// SIMATIC STEP 7 (V5.x) project GYPSUM
// CPU: CPU 317-2 DP
// station: P_ADR_BUS
// station: _S7H_BUSSYSTEM_CT
// station: Hardware
// station: SIMATIC 300(1)
// program: S7 Program(1)

SYMBOL_TABLE
"GROUPS"	DB 15	DB 15
"ROUTES"	DB 16	DB 16
"HMI"	DB 20	DB 20	// HMI
"RECEPT"	DB 21	DB 21
"G00_MILL_GYPSUM"	DB 30	FB 103	// Mill Gypsum
"G01_BIN_LOAD"	DB 31	FB 103	// 311BI100 Loading
"G02_EFILER"	DB 32	FB 103	// ElectroFilter Group
"G03_FRESH_GYPSUM"	DB 33	FB 103	// Fresh Gypsum
"G04_BOILER1"	DB 34	FB 103	// Boiler 1 Group
"G05_WEIGHT_PALLET"	DB 35	FB 103	// Weight Pallet
"G06_DISCHARGE"	DB 36	FB 103	// Discharge Group
"G07_BOILER2"	DB 37	FB 103	// G07 Boiler 2
"G08_BOILER3"	DB 38	FB 103	// G08 Boiler 3
"G17_DUMMY_LOCAL"	DB 47	FB 103
"G18_DUMMY_MANUAL"	DB 48	FB 103
"G19_DUMMY_ASTR"	DB 49	FB 103
"REG_T_BeforeSeparator"	DB 51	FB 41	// Temperature Regler Before Separator
"REG_DiffP_AfterSeparator"	DB 52	FB 41	// Diff Pressure Regler After Separator
"REG_Curr_CrusherMD140"	DB 53	FB 41	// Current Regler Crusher MD140
"REG_DiffP_Boiler3"	DB 54	FB 41	// Diff Pressure Regler Boiler  3
"REG_DiffP_Boiler1"	DB 55	FB 41	// Diff Pressure Regler Boiler 1
"REG_DiffP_Boiler2"	DB 56	FB 41	// Diff Pressure Regler Boiler 2
"Weight351BI100"	DB 61	FB 310	// Weight351BI100
"Weight351BI200"	DB 62	FB 310	// Weight351BI200
"Weight351BI300"	DB 63	FB 310	// Weight 351BI300 Fresh Gypsum
"Weight352BI100"	DB 64	FB 310	// Weight352BI100
"Weight352BI200"	DB 65	FB 310
"Weight352BI300"	DB 66	FB 310	// Weight352BI300
"Weight351BI130"	DB 67	FB 310	// Weight351BI130
"Weight351BI230"	DB 68	FB 310	// Weight351BI230
"Weight351BI330"	DB 69	FB 310	// Weight351BI330
"Boiler 1"	DB 70	FB 310	// Boler 1
"Boiler 2"	DB 71	FB 310	// Boiler 2
"Boiler 3"	DB 72	FB 310	// Boiler 3
"411DC100N01T01"	DB 101	FB 101	// Temperature Before Crusher
"411DC100N02P01"	DB 102	FB 101	// Pressure Before Crusher
"411DC100N03T02"	DB 103	FB 101	// Temperature After Crusher
"411DC100N04P02"	DB 104	FB 101	// Pressure After Crusher
"351BR300N06T04"	DB 105	FB 101	// Temperature Hot Air
"351BR300N07P03"	DB 106	FB 101	// Pressure Hot Air
"351BI100N01T01"	DB 107	FB 101	// Temperature In 351BI100
"351BI200N01T01"	DB 108	FB 101	// Temperature In 351BI200
"351BI300N01T01"	DB 109	FB 101	// Temperature In 351BI300
"351BR100N01T01"	DB 110	FB 101	// Temperature In Boiler 1 Top
"351BR100N02T02"	DB 111	FB 101	// Temperature In Boiler 1 Bottom
"351BR100N03P01"	DB 112	FB 101	// Pressure In Boiler 1 Bottom
"351BR200N01T01"	DB 113	FB 101	// Temperature In Boiler 2 Top
"351BR200N02T02"	DB 114	FB 101	// Temperature In Boiler 2 Bottom
"351BR200N03P01"	DB 115	FB 101	// Pressure In Boiler 2 Bottom
"351BR300N01T01"	DB 116	FB 101	// Temperature In Biler 3 Top
"351BR300N02T02"	DB 117	FB 101	// Temperature In Boiler 3 Bottom
"351BR300N03P01"	DB 118	FB 101	// Pressure In Boiler 3 Bottom
"331EP100N01P01"	DB 119	FB 101	// Pressure Before EFilter
"351BI100N02W01"	DB 120	FB 101	// Bin Weight 351BI100
"351BI200N02W01"	DB 121	FB 101	// Bin Weight 351BI200
"351BI300N02W01"	DB 122	FB 101	// Bin Weight 351BI300
"352BI100N01W01"	DB 123	FB 101	// Bin Weight 352BI100
"352BI200N01W01"	DB 124	FB 101	// Bin Weight 352BI200
"352BI300N01W01"	DB 125	FB 101	// Bin Weight 352BI300
"351BI130N01W01"	DB 126	FB 101	// Bin Weight 351BI130
"351BI230N01W01"	DB 127	FB 101	// Bin Weight 351BI230
"351BI330N01W01"	DB 128	FB 101	// Bin Weight 351BI330
"331EP100N02T01"	DB 129	FB 101	// Temperature Before EFilter
"331EP100N03T02"	DB 130	FB 101	// Temperature After EFilter
"331EP100N04P02"	DB 131	FB 101	// Pressure After EFilter
"331LD391Z01"	DB 132	FB 101	// Position Gate
"331LD392Z01"	DB 133	FB 101	// Position Gate
"411CN101N01P01"	DB 134	FB 101	// Pressure Before Cyclone
"411CN101N02T01"	DB 135	FB 101	// Temperature Before Cyclone
"411CN101N03P02"	DB 136	FB 101	// Pressure After Cyclone
"411CN101N04T02"	DB 137	FB 101	// Temperature After Cyclone
"411CN103N01P01"	DB 138	FB 101	// Pressure After Cyclone
"411CN103N02T01"	DB 139	FB 101	// Temperature After Cyclone
"351BR100N04T03"	DB 140	FB 101	// Temperature in Burner Boiler 1
"351BR100N05P02"	DB 141	FB 101	// Pressure In Burner Boiler 1
"351BR200N04T03"	DB 142	FB 101	// Temperature In Boiler 2
"351BR200N05P02"	DB 143	FB 101	// Pressure In Burner Boiler 2
"351BR300N04T03"	DB 144	FB 101	// Temperature In Burner Boiler 3
"351BR300N05P02"	DB 145	FB 101	// Pressure In Burner Boiler 3
"411SR150N03T02"	DB 146	FB 101	// Temperature Before Separator (Bearing)
"SPARE_AI47"	DB 147	FB 101
"143CV100SI01"	DB 148	FB 101	// Speed Chain Conveyor CV100
"143CV100UA01"	DB 149	FB 101	// Current Chain Conveyor CV100
"143BC200SI01"	DB 150	FB 101	// Speed Belt Conveyor BC200
"143BC200UA01"	DB 151	FB 101	// Current Belt Conveyor BC200
"331FN401SI01"	DB 152	FB 101	// Speed EFilter Fan FN401
"331FN401UA01"	DB 153	FB 101	// Current EFilter Fan FN401
"311TF150SI01"	DB 154	FB 101	// Speed Table Feeder TF150
"311TF150UA01"	DB 155	FB 101	// Current Table Feeder TF150
"411MD140SI01"	DB 156	FB 101	// Speed Crusher MD140
"411MD140UA01"	DB 157	FB 101	// Current Crusher MD140
"411MD152SI01"	DB 158	FB 101	// Speed Separator MD152
"411MD152UA01"	DB 159	FB 101	// Current Separator MD152
"351SC120SI01"	DB 160	FB 101	// Speed Screw Conveyor SC120
"351SC120UA01"	DB 161	FB 101	// Current Screw Conveyor SC120
"351SC220SI01"	DB 162	FB 101	// Speed Screw Conveyor SC220
"351SC220UA01"	DB 163	FB 101	// Current Screw Conveyor SC220
"351SC320SI01"	DB 164	FB 101	// Speed Screw Conveyor SC320
"351SC320UA01"	DB 165	FB 101	// Current Screw Conveyor SC320
"361SC140SI01"	DB 166	FB 101	// Speed Screw Conveyor SC140
"361SC140UA01"	DB 167	FB 101	// Current Screw Conveyor SC140
"351BR100N06T04"	DB 168	FB 101	// Temperature Hot Air From Boiler 1
"351BR200N06T04"	DB 169	FB 101	// Temperature Hot Air From Boiler 2
"351BR300N08T04"	DB 170	FB 101	// Temperature Hot Air From Boiler 3
"351SD101N01Z01"	DB 171	FB 101
"351SD102N01Z01"	DB 172	FB 101
"351SD103N01Z01"	DB 173	FB 101
"351SD104N01Z01"	DB 174	FB 101
"351Sd105N01Z01"	DB 175	FB 101
"100CP100N01P01"	DB 176	FB 101	// Pressure After Compressor
"BE120_CUR"	DB 177	FB 101	// BE120 Current AL
"SPARE_AI78"	DB 178	FB 101
"SPARE_AI79"	DB 179	FB 101
"SPARE_AI80"	DB 180	FB 101
"SPARE_AI81"	DB 181	FB 101
"SPARE_AI82"	DB 182	FB 101
"SPARE_AI83"	DB 183	FB 101
"SPARE_AI84"	DB 184	FB 101
"SPARE_AI85"	DB 185	FB 101
"SPARE_AI86"	DB 186	FB 101
"SPARE_AI87"	DB 187	FB 101
"SPARE_AI88"	DB 188	FB 101
"SPARE_AI89"	DB 189	FB 101
"SPARE_AI90"	DB 190	FB 101
"SPARE_AI91"	DB 191	FB 101
"SPARE_AI92"	DB 192	FB 101
"SPARE_AI93"	DB 193	FB 101
"SPARE_AI94"	DB 194	FB 101
"SPARE_AI95"	DB 195	FB 101
"SPARE_AI96"	DB 196	FB 101
"SPARE_AI97"	DB 197	FB 101
"SPARE_AI98"	DB 198	FB 101
"SPARE_AI99"	DB 199	FB 101
"SPARE_UNIMOTOR01"	DB 201	FB 110
"143BF120"	DB 202	FB 110	// Filter Control
"351VI110"	DB 203	FB 110	// Vibrator
"351VI210"	DB 204	FB 110	// Vibrator
"351VI310"	DB 205	FB 110	// Vibrator
"352VI110"	DB 206	FB 110	// Vibrator
"352VI111"	DB 207	FB 110	// Vibrator
"352VI210"	DB 208	FB 110	// Vibrator
"352VI211"	DB 209	FB 110	// Vibrator
"352VI310"	DB 210	FB 110	// Vibrator
"352VI311"	DB 211	FB 110	// Vibrator
"EP100P1"	DB 212	FB 110	// EFilter Pole 1
"EP100P2"	DB 213	FB 110	// EFilter Pole   2
"SPARE_UNIMOTOR14"	DB 214	FB 110
"SPARE_UNIMOTOR15"	DB 215	FB 110
"SPARE_UNIMOTOR16"	DB 216	FB 110
"SPARE_UNIMOTOR17"	DB 217	FB 110
"SPARE_UNIMOTOR18"	DB 218	FB 110
"SPARE_UNIMOTOR19"	DB 219	FB 110
"SPARE_UNIMOTOR20"	DB 220	FB 110
"411SD311"	DB 251	FB 102	// Gate Gypsum To Pneumatic Pump
"412SD321"	DB 252	FB 102	// Gate Gypsum To Screw Conveyor
"411SD331"	DB 253	FB 102	// Gate Weight 351BI100 Inlet
"411SD332"	DB 254	FB 102	// Gate Weight 351BI200 Inlet
"411SD333"	DB 255	FB 102	// Gate Weight 351BI300 Inlet
"351SD140"	DB 256	FB 102	// Gate Boiler 1 Outlet
"351SD141"	DB 257	FB 102	// Gate Boiler 1 Outlet
"352SD120"	DB 258	FB 102	// Gate Weight 352BI100 Outlet
"352SD121"	DB 259	FB 102	// Gate Weight 352BI100 Outlet
"351SD240"	DB 260	FB 102	// Gate Boiler 2 Outlet
"351SD241"	DB 261	FB 102	// Gate Boiler 2 Outlet
"352SD220"	DB 262	FB 102	// Gate Weight 352BI200 Outlet
"352SD221"	DB 263	FB 102	// Gate Weight 352BI200 Outlet
"351SD340"	DB 264	FB 102	// Gate Boiler 3 Outlet
"351SD341"	DB 265	FB 102	// Gate Boiler 3 Outlet
"352SD320"	DB 266	FB 102	// Gate Weight 352BI300 Outlet
"352SD321"	DB 267	FB 102	// Gate Weight 352BI300 Outlet
"361SD170"	DB 268	FB 102	// Gate 371BI500 Inlet
"361SD171"	DB 269	FB 102	// Gate 371BI100 Inlet
"361SD172"	DB 270	FB 102	// Gate 371BI100 Inlet
"361SD173"	DB 271	FB 102	// Gate 371BI200 Inlet
"361SD174"	DB 272	FB 102	// Gate 371B200 Inlet
"361SD175"	DB 273	FB 102	// Gate 371BI300 Inlet
"361SD176"	DB 274	FB 102	// Gate 371BI300 Inlet
"361SD177"	DB 275	FB 102	// Gate 371BI400 Inlet
"351BV031"	DB 276	FB 102	// Valve Aqua To Boiler 1
"351BV032"	DB 277	FB 102	// Valve Aqua To Boiler 2
"351BV033"	DB 278	FB 102	// Valve Aqua To Boiler 3
"351SD135"	DB 279	FB 102	// Gate Weight 351BI130 Inlet
"351SD235"	DB 280	FB 102	// Gate Weight 351BI230 Inlet
"351SD335"	DB 281	FB 102	// Gate Weight 351BI330 Inlet
"411BV151"	DB 282	FB 102	// Valve Separator Aspiration
"SPARE_VALVE33"	DB 283	FB 102
"351SD106"	DB 284	FB 102	// Gate Boiler 1 Outlet Hot Air
"351SD107"	DB 285	FB 102	// Gate Boiler 1 Outlet
"351SD108"	DB 286	FB 102	// Gate Boiler 3 Outlet
"351SD109"	DB 287	FB 102	// Gate Hot Air To Gypsum Line
"SPARE_VALVE38"	DB 288	FB 102
"SPARE_VALVE39"	DB 289	FB 102
"SPARE_VALVE40"	DB 290	FB 102
"SPARE_UMOTSC01"	DB 301	FB 134
"143VF150"	DB 302	FB 134	// Vibrating Din
"143BC160"	DB 303	FB 134	// Belt Conveyor
"SPARE_UMOTSC04"	DB 304	FB 134
"143RB250"	DB 305	FB 134	// Crusher
"143BE300"	DB 306	FB 134	// Elevator
"143FN122"	DB 307	FB 134	// Filter Fan
"311RF200"	DB 308	FB 134	// Rotary Feeder
"41FN101"	DB 309	FB 134	// Fan Crusher Drive Cooling
"411RF201"	DB 310	FB 134	// Rotary Feeder
"411RF304"	DB 311	FB 134	// Rotary Feeder
"411SC322"	DB 312	FB 134	// Screw Conveyor
"331VI201"	DB 313	FB 134	// Filter Rapping 1
"331VI202"	DB 314	FB 134	// Filter Rapping 2
"331VI203"	DB 315	FB 134	// Filter Rapping 3
"331VI204"	DB 316	FB 134	// Filter Rapping 4
"331RF301"	DB 317	FB 134	// Rotary Feeder
"331RF302"	DB 318	FB 134	// Rotary Feeder
"331RF303"	DB 319	FB 134	// Rotary Feeder
"331SC351"	DB 320	FB 134	// Screw Conveyor
"411RF314"	DB 321	FB 134	// Rotary Feeder
"361SC150"	DB 322	FB 134	// Screw Conveyor
"SPARE_UMOTSC23"	DB 323	FB 134
"411PP312"	DB 324	FB 134	// Pneumatic Pump
"SPARE_UMOTSC25"	DB 325	FB 134
"SPARE_UMOTSC26"	DB 326	FB 134
"351AG130"	DB 327	FB 134	// Mixer 1
"351AG230"	DB 328	FB 134	// Mixer 2
"351AG330"	DB 329	FB 134	// Mixer 3
"361SC110"	DB 330	FB 134	// Screw Conveyor
"361SC111"	DB 331	FB 134	// Screw Conveyor
"361BE120"	DB 332	FB 134	// Elevator
"361SC130"	DB 333	FB 134	// Screw Conveyor
"SPARE_UMOTSC34"	DB 334	FB 134
"361SC141"	DB 335	FB 134	// Screw Conveyor
"SPARE_UMOTSC36"	DB 336	FB 134
"361SC160"	DB 337	FB 134	// Screw Conveyor
"341RF101"	DB 338	FB 134	// Rotary Feeder
"SPARE_UMOTSC39"	DB 339	FB 134	// Spare
"411FN200"	DB 340	FB 134	// Fan Hot Air To Crusher
"351AG050"	DB 341	FB 134	// Mixer
"351SP100"	DB 342	FB 134	// Pump
"SPARE_UMOTSC43"	DB 343	FB 134
"SPARE_UMOTSC44"	DB 344	FB 134
"SPARE_UMOTSC45"	DB 345	FB 134
"SPARE_UMOTSC46"	DB 346	FB 134
"SPARE_UMOTSC47"	DB 347	FB 134
"SPARE_UMOTSC48"	DB 348	FB 134
"SPARE_UMOTSC49"	DB 349	FB 134
"SPARE_UMOTSC50"	DB 350	FB 134
"SPARE_UMOTSC51"	DB 351	FB 134
"SPARE_UMOTSC52"	DB 352	FB 134
"SPARE_UMOTSC53"	DB 353	FB 134
"SPARE_UMOTSC54"	DB 354	FB 134
"SPARE_UMOTSC55"	DB 355	FB 134
"SPARE_UMOTSC56"	DB 356	FB 134
"SPARE_UMOTSC57"	DB 357	FB 134
"SPARE_UMOTSC58"	DB 358	FB 134
"SPARE_UMOTSC59"	DB 359	FB 134
"SPARE_UMOTSC60"	DB 360	FB 134
"SPARE_UMOTSC61"	DB 361	FB 134
"SPARE_UMOTSC62"	DB 362	FB 134
"SPARE_UMOTSC63"	DB 363	FB 134
"SPARE_UMOTSC64"	DB 364	FB 134
"SPARE_UMOTSC65"	DB 365	FB 134
"SPARE_UMOTSC66"	DB 366	FB 134
"SPARE_UMOTSC67"	DB 367	FB 134
"SPARE_UMOTSC68"	DB 368	FB 134
"SPARE_UMOTSC69"	DB 369	FB 134
"SPARE_UMOTSC70"	DB 370	FB 134
"SPARE_UMOTSC71"	DB 371	FB 134
"SPARE_UMOTSC72"	DB 372	FB 134
"SPARE_UMOTSC73"	DB 373	FB 134
"SPARE_UMOTSC74"	DB 374	FB 134
"SPARE_UMOTSC75"	DB 375	FB 134
"SPARE_UMOTSC76"	DB 376	FB 134
"SPARE_UMOTSC77"	DB 377	FB 134
"SPARE_UMOTSC78"	DB 378	FB 134
"SPARE_UMOTSC79"	DB 379	FB 134
"SPARE_UMOTSC80"	DB 380	FB 134
"SPARE_UMOTSC81"	DB 381	FB 134
"SPARE_UMOTSC82"	DB 382	FB 134
"SPARE_UMOTSC83"	DB 383	FB 134
"SPARE_UMOTSC84"	DB 384	FB 134
"SPARE_UMOTSC85"	DB 385	FB 134
"SPARE_UMOTSC86"	DB 386	FB 134
"SPARE_UMOTSC87"	DB 387	FB 134
"SPARE_UMOTSC88"	DB 388	FB 134
"SPARE_UMOTSC89"	DB 389	FB 134
"SPARE_UMOTSC90"	DB 390	FB 134
"SPARE_UMOTSC91"	DB 391	FB 134
"SPARE_UMOTSC92"	DB 392	FB 134
"SPARE_UMOTSC93"	DB 393	FB 134
"SPARE_UMOTSC94"	DB 394	FB 134
"SPARE_UMOTSC95"	DB 395	FB 134
"SPARE_UMOTSC96"	DB 396	FB 134
"SPARE_UMOTSC97"	DB 397	FB 134
"SPARE_UMOTSC98"	DB 398	FB 134
"SPARE_UMOTSC99"	DB 399	FB 134
"331LD391_SPARE"	DB 401	FB 136	// Gate Filter Fan
"331LD392_SPARE"	DB 402	FB 136	// Gate Filter Fan
"SPARE_AGATESC03"	DB 403	FB 136
"SPARE_AGATESC04"	DB 404	FB 136
"SPARE_AGATESC05"	DB 405	FB 136
"SPARE_AGATESC06"	DB 406	FB 136
"SPARE_AGATESC07"	DB 407	FB 136
"SPARE_AGATESC08"	DB 408	FB 136
"SPARE_AGATESC09"	DB 409	FB 136
"SPARE_AGATESC10"	DB 410	FB 136
"SPARE_GATESC01"	DB 451	FB 135
"SPARE_GATESC02"	DB 452	FB 135
"SPARE_GATESC03"	DB 453	FB 135
"SPARE_GATESC04"	DB 454	FB 135
"SPARE_GATESC05"	DB 455	FB 135
"SPARE_GATESC06"	DB 456	FB 135
"SPARE_GATESC07"	DB 457	FB 135
"SPARE_GATESC08"	DB 458	FB 135
"SPARE_GATESC09"	DB 459	FB 135
"SPARE_GATESC10"	DB 460	FB 135
"SPARE_BIMOTSC01"	DB 501	FB 139
"SPARE_BIMOTSC02"	DB 502	FB 139
"SPARE_BIMOTSC03"	DB 503	FB 139
"SPARE_BIMOTSC04"	DB 504	FB 139
"SPARE_BIMOTSC05"	DB 505	FB 139
"SPARE_BIMOTSC06"	DB 506	FB 139
"SPARE_BIMOTSC07"	DB 507	FB 139
"SPARE_BIMOTSC08"	DB 508	FB 139
"SPARE_BIMOTSC09"	DB 509	FB 139
"SPARE_BIMOTSC10"	DB 510	FB 139
"SPARE_BIMOTOR01"	DB 551	FB 109
"SPARE_BIMOTOR02"	DB 552	FB 109
"SPARE_BIMOTOR03"	DB 553	FB 109
"SPARE_BIMOTOR04"	DB 554	FB 109
"SPARE_BIMOTOR05"	DB 555	FB 109
"SPARE_BIMOTOR06"	DB 556	FB 109
"SPARE_BIMOTOR07"	DB 557	FB 109
"SPARE_BIMOTOR08"	DB 558	FB 109
"SPARE_BIMOTOR09"	DB 559	FB 109
"SPARE_BIMOTOR10"	DB 560	FB 109
"331FN401"	DB 601	FB 111	// Fan EP Filter
"411MD140"	DB 602	FB 111	// Crusher
"311TF150"	DB 603	FB 111	// Table Feeder
"411MD152"	DB 604	FB 111	// Separator
"143BC200"	DB 605	FB 111	// Belt Conveyor
"361SC140"	DB 606	FB 111	// Screw Conveyor
"143CV100"	DB 607	FB 111	// Chain conveyor
"351SC120"	DB 608	FB 111	// Screw Conveyor
"351SC220"	DB 609	FB 111	// Screw Conveyor
"351SC320"	DB 610	FB 111	// Screw Conveyor
"SPARE_FC11"	DB 611	FB 111
"SPARE_FC12"	DB 612	FB 111
"WF_GROUP"	DB 650	FB 50
"SPARE_WF01"	DB 651	FB 50
"SPARE_WF02"	DB 652	FB 50
"SPARE_WF03"	DB 653	FB 50
"SPARE_WF04"	DB 654	FB 50
"SPARE_WF05"	DB 655	FB 50
"SPARE_WF06"	DB 656	FB 50
"SPARE_WF07"	DB 657	FB 50
"SPARE_WF08"	DB 658	FB 50
"SPARE_WF09"	DB 659	FB 50
"SPARE_WF10"	DB 660	FB 50
"SERV_VALVE"	DB 700	DB 700	// Service VALVE
"SERV_UMOT"	DB 701	DB 701	// SERVICE UNIMOTOR
"SERV_FC"	DB 702	DB 702	// SERVICE FC
"SERV_POSITIONER"	DB 703	DB 703	// SERVICE POSITIONER
"SERV_ANALOG"	DB 704	DB 704	// SERVICE ANALOG
"SERV_GATE"	DB 705	DB 705
"SERV_AGATE"	DB 706	DB 706
"SERV_BIMOT"	DB 709	DB 709
"SERV_UMOT_SC"	DB 710	DB 710	// SERVICE UNIMOTOR_SC
"SERV_BIMOT_SC"	DB 711	DB 711	// SERVICE BIMOT_SC
"SERV_GATE_SC"	DB 712	DB 712	// SERVICE GATE_SC
"SERV_AGATE_SC"	DB 714	DB 714	// SERVICE AGATE_SC
"SERV_WF"	DB 715	DB 715	// SERVICE WF
"SPARE_GATE01"	DB 751	FB 105
"SPARE_GATE02"	DB 752	FB 105
"SPARE_GATE03"	DB 753	FB 105
"SPARE_GATE04"	DB 754	FB 105
"SPARE_GATE05"	DB 755	FB 105
"SPARE_AGATE01"	DB 771	FB 106
"SPARE_AGATE02"	DB 772	FB 106
"SPARE_AGATE03"	DB 773	FB 106
"SPARE_AGATE04"	DB 774	FB 106
"SPARE_AGATE05"	DB 775	FB 106
"BE300_LEVEL_MAX"	DB 801	FB 151	// Elevator BE300 Level Max Alarm
"311BI100_LEVEL_H"	DB 802	FB 151	// 311BI100 Level Max Alarm
"311BI100_LEVEL_L"	DB 803	FB 151	// 311BI100 Level Min Alarm
"371BI100_LEVEL_H"	DB 804	FB 151	// 371BI100 Level Max Alarm
"371BI100_LEVEL_L"	DB 805	FB 151	// 371BI100 Level Min Alarm
"371BI200_LEVEL_H"	DB 806	FB 151	// 371BI200 Level Max Alarm
"371BI200_LEVEL_L"	DB 807	FB 151	// 371BI200 Level Min Alarm
"371BI300_LEVEL_H"	DB 808	FB 151	// 371BI300 Level Max Alarm
"371BI300_LEVEL_L"	DB 809	FB 151	// 371BI300 Level Min Alarm
"371BI400_LEVEL_H"	DB 810	FB 151	// 371BI400 Level Max Alarm
"371BI400_LEVEL_L"	DB 811	FB 151	// 371BI400 Level Min Alarm
"371BI500_LEVEL_H"	DB 812	FB 151	// 371BIN500 Level Max Alarm
"371BI500_LEVEL_L"	DB 813	FB 151	// 371BIN500 Level Min Alarm
"BE120_LEVEL_H"	DB 814	FB 151	// Elevator BE120 Level Max Alarm
"341BI100_LEVEL_H"	DB 815	FB 151	// 341BI100 Level Max Alarm
"341BI100_LEVEL_L"	DB 816	FB 151	// 341BI100 Level Min Alarm
"311FN401_SELECTED"	DB 817	FB 151	// FN401 Selected
"311FN402_SELECTED"	DB 818	FB 151	// FN402 Selected
"441BI100_LEVEL_H"	DB 819	FB 151	// 441BI100 Level Max Alarm
"441BI100_LEVEL_L"	DB 820	FB 151	// 441BI100 Level Min Alarm
"FA2_380V"	DB 821	FB 151	// Circuit switch 380 VAC - SITOP
"FA22_220V"	DB 822	FB 151	// Circuit switch 220 VAC - Valve 1
"K3UPS"	DB 823	FB 151	// Voltage before UPS - 220 VAC
"FA20_220V"	DB 824	FB 151	// Circuit switch 220 VAC - Main voltage
"FA3_24V"	DB 825	FB 151	// Circuit switch 24 VDC - MCC Main voltage
"FA31_24V"	DB 826	FB 151	// Circuit switch 24 VDC - Main voltage
"FA40_24V"	DB 827	FB 151	// Circuit switch 24 VDC - DO Moduls A7, A8
"FA41_24V"	DB 828	FB 151	// Circuit switch 24 VDC - AI Modul A12
"FA42_24V"	DB 829	FB 151	// Circuit switch 24 VDC - AI Modul A13
"FA43_24V"	DB 830	FB 151	// Circuit switch 24 VDC - AI Modul A14
"FA44_24V"	DB 831	FB 151	// Circuit switch 24 VDC - AI Modul A15
"FA45_24V"	DB 832	FB 151	// Circuit switch 24 VDC - AI Modul A16
"FA46_24V"	DB 833	FB 151	// Circuit switch 24 VDC - AI Modul A17
"FA47_24V"	DB 834	FB 151	// Circuit switch 24 VDC - AO Modul A18
"FA23_220V"	DB 835	FB 151	// Circuit switch 220 VAC - Valve 2
"SR_OK"	DB 836	FB 151	// Safety Rellay OK
"FA24_220V"	DB 837	FB 151	// Circuit switch 220 VAC - Light control and Horn
"FA25_220V"	DB 838	FB 151	// Circuit switch 220 VAC - Level MIKMA
"FA48_24V"	DB 839	FB 151	// Circuit switch 24 VDC - AI Modul A19
"EF_DISCH_EN"	DB 840	FB 151	// EFilter Discharge Enable
"EF_BIGBAG_FULL"	DB 841	FB 151	// EFilter Big Bag Full
"SPARE_ALARM42"	DB 842	FB 151
"SPARE_ALARM43"	DB 843	FB 151
"SPARE_ALARM44"	DB 844	FB 151
"SPARE_ALARM45"	DB 845	FB 151
"SPARE_ALARM46"	DB 846	FB 151
"SPARE_ALARM47"	DB 847	FB 151
"SPARE_ALARM48"	DB 848	FB 151
"SPARE_ALARM49"	DB 849	FB 151
"SPARE_ALARM50"	DB 850	FB 151
"SPARE_ALARM51"	DB 851	FB 151
"SPARE_ALARM52"	DB 852	FB 151
"SPARE_ALARM53"	DB 853	FB 151
"SPARE_ALARM54"	DB 854	FB 151
"SPARE_ALARM55"	DB 855	FB 151
"SPARE_ALARM56"	DB 856	FB 151
"SPARE_ALARM57"	DB 857	FB 151
"SPARE_ALARM58"	DB 858	FB 151
"SPARE_ALARM59"	DB 859	FB 151
"SPARE_ALARM60"	DB 860	FB 151
"SPARE_ALARM61"	DB 861	FB 151
"SPARE_ALARM62"	DB 862	FB 151
"SPARE_ALARM63"	DB 863	FB 151
"SPARE_ALARM64"	DB 864	FB 151
"SPARE_ALARM65"	DB 865	FB 151
"SPARE_ALARM66"	DB 866	FB 151
"SPARE_ALARM67"	DB 867	FB 151
"SPARE_ALARM68"	DB 868	FB 151
"SPARE_ALARM69"	DB 869	FB 151
"SPARE_ALARM70"	DB 870	FB 151
"SPARE_ALARM71"	DB 871	FB 151
"SPARE_ALARM72"	DB 872	FB 151
"SPARE_ALARM73"	DB 873	FB 151
"SPARE_ALARM74"	DB 874	FB 151
"SPARE_ALARM75"	DB 875	FB 151
"SPARE_ALARM76"	DB 876	FB 151
"SPARE_ALARM77"	DB 877	FB 151
"SPARE_ALARM78"	DB 878	FB 151
"SPARE_ALARM79"	DB 879	FB 151
"SPARE_ALARM80"	DB 880	FB 151
"SPARE_ALARM81"	DB 881	FB 151
"SPARE_ALARM82"	DB 882	FB 151
"SPARE_ALARM83"	DB 883	FB 151
"SPARE_ALARM84"	DB 884	FB 151
"SPARE_ALARM85"	DB 885	FB 151
"SPARE_ALARM86"	DB 886	FB 151
"SPARE_ALARM87"	DB 887	FB 151
"SPARE_ALARM88"	DB 888	FB 151
"SPARE_ALARM89"	DB 889	FB 151
"SPARE_ALARM90"	DB 890	FB 151
"SPARE_ALARM91"	DB 891	FB 151
"SPARE_ALARM92"	DB 892	FB 151
"SPARE_ALARM93"	DB 893	FB 151
"SPARE_ALARM94"	DB 894	FB 151
"SPARE_ALARM95"	DB 895	FB 151
"SPARE_ALARM96"	DB 896	FB 151
"SPARE_ALARM97"	DB 897	FB 151
"SPARE_ALARM98"	DB 898	FB 151
"SPARE_ALARM99"	DB 899	FB 151
"FN401_SELECT"	DB 901	FB 108	// Select FN401
"FN402_SELECT"	DB 902	FB 108	// Select FN402
"NO_VIBDIN_SELECT"	DB 903	FB 108	// Without Vibrating Din Select
"CRUSHER_LOAD_EN"	DB 904	FB 108	// Crusher Load Eanble
"411PP312_ SELECT"	DB 905	FB 108	// Gypsum To Line 1
"351BI100_SELECT"	DB 906	FB 108	// 351BI100 Select
"351BI200_SELECT"	DB 907	FB 108	// 351BI200 Select
"351BI300_SELECT"	DB 908	FB 108	// 351BI300 Select
"BOILER1_LOAD_EN"	DB 909	FB 108	// Boiler 1 Load Enable
"BOILER2_LOAD_EN"	DB 910	FB 108	// Boiler 2 Load Enable
"BOILER3_LOAD_EN"	DB 911	FB 108	// Boiler 3 Load Eanble
"352SD120_SELECT"	DB 912	FB 108	// 352SD120 Select
"352SD220_SELECT"	DB 913	FB 108	// 352SD220_SELECT
"352SD320_SELECT"	DB 914	FB 108	// 352SD320_SELECT
"361SD170_SELECT"	DB 915	FB 108	// 361SD170 Select Load To Bin500
"361SD171_SELECT"	DB 916	FB 108	// 361SD171 Select Load To Bin100
"361SD172_SELECT"	DB 917	FB 108	// 361SD172 Select Load To Bin100
"361SD173_SELECT"	DB 918	FB 108	// 361SD173 Select Load To Bin 200
"361SD174_SELECT"	DB 919	FB 108	// 361SD174 Select Load To Bin 200
"361SD175_SELECT"	DB 920	FB 108	// 361SD175 Select Load To Bin 300
"361SD176_SELECT"	DB 921	FB 108	// 361SD176 Select Load To Bin 300
"361SD177_SELECT"	DB 922	FB 108	// 361SD177 Select Load To Bin 400
"352SD121_SELECT"	DB 923	FB 108	// 352SD121_SELECT
"352SD221_SELECT"	DB 924	FB 108	// 352SD221_SELECT
"352SD321_SELECT"	DB 925	FB 108	// 352SD321_SELECT
"REG_T_BS_AUT_SLELECT"	DB 926	FB 108	// Regler Auto manual mode Select
"361SC111_SELECT"	DB 927	FB 108
"REG_DiffPSepar_SELECT"	DB 928	FB 108	// Regler Diff Pressur After Separator Select
"REG_Curr_MD140_SELECT"	DB 929	FB 108	// Regler Current MD140 Select
"REG_DiffP_Boiler3_SELECT"	DB 930	FB 108	// Regler Diff Pressure Boiler 3 Selecct
"REG_DiffP_Boiler1_SELECT"	DB 931	FB 108	// Regler Diff Pressure Boiler 1
"REG_DiffP_Boiler2_SELECT"	DB 932	FB 108	// Regler Diff Pressure Boiler 2 Select
"SPARE_SELECT33"	DB 933	FB 108
"411SD301"	DB 1001	FB 115	// Positioner Cyclone CN100 Outlet
"411SD302"	DB 1002	FB 115	// Positioner Cyclone CN101 Outlet
"351SD101"	DB 1003	FB 115	// Positioner Boiler 1 Outlet
"351SD102"	DB 1004	FB 115	// Positioner Boiler 2 Outlet
"351SD103"	DB 1005	FB 115	// Positioner Boiler 3 Outlet
"351SD104_"	DB 1006	FB 115	// AGATE Fresh Air
"351SD105_"	DB 1007	FB 115	// PosGate
"CONT_C"	FB 41	FB 41	// Continuous Control
"WEIGHTFEEDER"	FB 50	FB 50	// WEICHT FEEDER
"REG_LINE2P"	FB 51	FB 51
"PLC1_PUT_GET"	FB 100	FB 100
"AI"	FB 101	FB 101
"VALVE"	FB 102	FB 102	// Valve
"GROUP"	FB 103	FB 103	// Group
"MAIN DRIVE"	FB 104	FB 104	// Main Drive
"GATE"	FB 105	FB 105	// GATE
"AGATE"	FB 106	FB 106	// AGATE
"ROUTE"	FB 107	FB 107
"SELECT"	FB 108	FB 108
"BIMOTOR"	FB 109	FB 109	// Rev Drive
"UNIMOTOR"	FB 110	FB 110
"FC"	FB 111	FB 111	// FC
"POSITIONER"	FB 115	FB 115	// POSITIONER
"UMOT_SC"	FB 134	FB 134	// UNIMOTOR_SC
"GATE_SC"	FB 135	FB 135	// MOTORGATE_SC
"AGATE_SC"	FB 136	FB 136	// AGATE_SC
"BIMOT_SC"	FB 139	FB 139	// BIMOT_SC
"ALARM"	FB 151	FB 151
"FEEDER"	FB 310	FB 310
"_HMI"	FC 20	FC 20	// HMI
"_SERVICE"	FC 25	FC 25	// SERVICE
"_G00_MILL_GYPSUM"	FC 30	FC 30
"_G01_BIN_LOAD"	FC 31	FC 31
"_G02_EFILTER"	FC 32	FC 32	// ElectroFilter
"_G03_FRESH_GYPSUM"	FC 33	FC 33
"_G04_BOILER1"	FC 34	FC 34
"_G05_WEIGHTS_PALLET"	FC 35	FC 35
"_G06_DISCHARGE"	FC 36	FC 36
"_G07_BOILER2"	FC 37	FC 37	// G07  Boler 2
"_G08_BOILER3"	FC 38	FC 38
"_G17_DLOCAL"	FC 47	FC 47	// DUMMY LOCAL
"_G18_DMANUAL"	FC 48	FC 48	// DUMMY MANUAL
"_G19_DASTR"	FC 49	FC 49	// DUMMY AUTO STR
"_SIM"	FC 55	FC 55	// Simulation
"_Weight351BI100"	FC 61	FC 61	// Bin Weight 351BI100
"_Weight351BI200"	FC 62	FC 62	// Bin Weight 351BI200
"_Weight351BI300"	FC 63	FC 63	// Bin Weight 351BI300
"_Weight352BI100"	FC 64	FC 64	// Bin Weight 352BI100
"_Weight352BI200"	FC 65	FC 65	// Bin Weight 352BI200
"_Weight352BI300"	FC 66	FC 66	// Bin Weigt 352BI300
"_Weight351BI130"	FC 67	FC 67	// Bin Weight Pallets
"_Weight351BI230"	FC 68	FC 68	// Bin Weight 351BI230
"_Weight351BI330"	FC 69	FC 69	// Bin Weight Pallets
"_Boiler 1"	FC 70	FC 70	// Boler 1 BR100
"_Boiler 2"	FC 71	FC 71	// Boiler 2 BR200
"_Boiler 3"	FC 72	FC 72	// Boiler 3 BR300
"_411DC100N01T01"	FC 101	FC 101	// Temperature Before Crusher
"_411DC100N02P01"	FC 102	FC 102	// Pressure Before Crusher
"_411DC100N03T02"	FC 103	FC 103	// Temperature After Crusher
"_411DC100N04P02"	FC 104	FC 104	// Pressure After Crusher
"_351BR300N06T04"	FC 105	FC 105	// Temperature Hot Air
"_351BR300N07P03"	FC 106	FC 106	// Pressure Hot Air
"_351BI100N01T01"	FC 107	FC 107	// Temperature In 351BI100
"_351BI200N01T01"	FC 108	FC 108	// Temperature In 351BI200
"_351BI300N01T01"	FC 109	FC 109	// Temperature In 351BI300
"_351BR100N01T01"	FC 110	FC 110	// Temperature In Boiler 1 Top
"_351BR100N02T02"	FC 111	FC 111	// Temperature In Boiler 1 Bottom
"_351BR100N03P01"	FC 112	FC 112	// Pressure In Boiler 1 Bottom
"_351BR200N01T01"	FC 113	FC 113	// Temperature In Boiler 2 Top
"_351BR200N02T02"	FC 114	FC 114	// Temperature In Boiler 2 Bottom
"_351BR200N03P01"	FC 115	FC 115	// Pressure In Boiler 2 Bottom
"_351BR300N01T01"	FC 116	FC 116	// Temperature In Boiler 3 Top
"_351BR300N02T02"	FC 117	FC 117	// Temperature In Boiler 3 Bottom
"_351BR300N03P01"	FC 118	FC 118	// Pressure In Boiler 3 Bottom
"_331EP100N01P01"	FC 119	FC 119	// Pressure Before EFilter
"_351BI100N02W01"	FC 120	FC 120	// Bin Weight 351BI100
"_351BI200N02W01"	FC 121	FC 121	// Bin Weight 351BI200
"_351BI300N02W01"	FC 122	FC 122	// Bin Weight 351BI300
"_352BI100N01W01"	FC 123	FC 123	// Bin Weight 352BI100
"_352BI200N01W01"	FC 124	FC 124	// Bin Weight 352BI200
"_352BI300N01W01"	FC 125	FC 125	// Bin Weight 352BI300
"_351BI130N01W01"	FC 126	FC 126	// Bin Weight 351BI130
"_351BI230N01W01"	FC 127	FC 127	// Bin Weight 351BI230
"_351BI330N01W01"	FC 128	FC 128	// Bin Weight 351BI330
"_331EP100N02T01"	FC 129	FC 129	// Temperature Before EFilter
"_331EP100N03T02"	FC 130	FC 130	// Temperature After EFilter
"_331EP100N04P02"	FC 131	FC 131	// Pressure After EFilter
"_331LD391Z01"	FC 132	FC 132	// Position Gate
"_331LD392Z01"	FC 133	FC 133	// Position Gate
"_411CN101N01P01"	FC 134	FC 134	// Pressure Before Cyclone
"_411CN101N02T01"	FC 135	FC 135	// Temperature Before Cyclone
"_411CN101N03P02"	FC 136	FC 136	// Pressure After Cyclone
"_411CN101N04T02"	FC 137	FC 137	// Temperature After Cyclone
"_411CN103N01P01"	FC 138	FC 138	// Pressure After Cyclone
"_411CN103N02T01"	FC 139	FC 139	// Temperature After Cyclone
"_351BR100N04T03"	FC 140	FC 140	// Temperature in Burner Boiler 1
"_351BR100N05P02"	FC 141	FC 141	// Pressure in Burner Boiler 1
"_351BR200N04T03"	FC 142	FC 142	// Temperature in Burner Boiler 2
"_351BR200N05P02"	FC 143	FC 143	// Pressure in Burner Boiler 2
"_351BR300N04T03"	FC 144	FC 144	// Temperature in Burner Boiler 3
"_351BR300N05P02"	FC 145	FC 145	// Pressure in Burner Boiler 3
"_411SR150N03T02"	FC 146	FC 146	// Temperature Before Separator (Bearing)
"_SPARE_AI47"	FC 147	FC 147
"_143CV100SI01"	FC 148	FC 148	// Speed Chain Conveyor CV100
"_143CV100UA01"	FC 149	FC 149	// Current Chain Conveyor CV100
"_143BC200SI01"	FC 150	FC 150	// Speed Belt Conveyor BC200
"_143BC200UA01"	FC 151	FC 151	// Current Belt Conveyor BC200
"_331FN401SI01"	FC 152	FC 152	// Speed EFilter Fan FN401
"_331FN401UA01"	FC 153	FC 153	// Current EFilter Fan FN401
"_311TF150SI01"	FC 154	FC 154	// Speed Table Feeder TF150
"_311TF150UA01"	FC 155	FC 155	// Current Table Feeder TF150
"_411MD140SI01"	FC 156	FC 156	// Speed Crusher MD140
"_411MD140UA01"	FC 157	FC 157	// Current Crusher MD140
"_411MD152SI01"	FC 158	FC 158	// Speed Separator MD152
"_411MD152UA01"	FC 159	FC 159	// Current Separator MD152
"_351SC120SI01"	FC 160	FC 160	// Speed Screw Conveyor SC120
"_351SC120UA01"	FC 161	FC 161	// Current Screw Conveyor SC120
"_351SC220SI01"	FC 162	FC 162	// Speed Screw Conveyor SC220
"_351SC220UA01"	FC 163	FC 163	// Current Screw Conveyor SC220
"_351SC320SI01"	FC 164	FC 164	// Speed Screw Conveyor SC320
"_351SC320UA01"	FC 165	FC 165	// Current Screw Conveyor SC320
"_361SC140SI01"	FC 166	FC 166	// Speed Screw Conveyor SC140
"_361SC140UA01"	FC 167	FC 167	// Current Screw Conveyor SC140
"_351BR100N06T04"	FC 168	FC 168	// Temperature Hot Air From Boiler 1
"_351BR200N06T04"	FC 169	FC 169	// Temperature Hot Air From Boiler 2
"_351BR300N08T04"	FC 170	FC 170	// Temperature Hot Air From Boiler 3
"_351SD101N01Z01"	FC 171	FC 171
"_351SD102N01Z01"	FC 172	FC 172
"_351SD103N01Z01"	FC 173	FC 173
"_351SD104N01Z01"	FC 174	FC 174
"_351SD105N01Z01"	FC 175	FC 175
"_100CP100N01P01"	FC 176	FC 176	// Pressure After Compressor
"_BE120_CUR"	FC 177	FC 177
"_SPARE_AI78"	FC 178	FC 178
"_SPARE_AI79"	FC 179	FC 179
"_SPARE_AI80"	FC 180	FC 180
"_SPARE_AI81"	FC 181	FC 181
"_SPARE_AI82"	FC 182	FC 182
"_SPARE_AI83"	FC 183	FC 183
"_SPARE_AI84"	FC 184	FC 184
"_SPARE_AI85"	FC 185	FC 185
"_SPARE_AI86"	FC 186	FC 186
"_SPARE_AI87"	FC 187	FC 187
"_SPARE_AI88"	FC 188	FC 188
"_SPARE_AI89"	FC 189	FC 189
"_SPARE_AI90"	FC 190	FC 190
"_SPARE_AI91"	FC 191	FC 191
"_SPARE_AI92"	FC 192	FC 192
"_SPARE_AI93"	FC 193	FC 193
"_SPARE_AI94"	FC 194	FC 194
"_SPARE_AI95"	FC 195	FC 195
"_SPARE_AI96"	FC 196	FC 196
"_SPARE_AI97"	FC 197	FC 197
"_SPARE_AI98"	FC 198	FC 198
"_SPARE_AI99"	FC 199	FC 199
"_SPARE_UNIMOTOR01"	FC 201	FC 201
"_143BF120"	FC 202	FC 202	// Fiilter Control
"_351VI110"	FC 203	FC 203	// Vibrator
"_351VI210"	FC 204	FC 204	// Vibrator
"_351VI310"	FC 205	FC 205	// Vibrator
"_352VI110"	FC 206	FC 206	// Vibrator
"_352VI111"	FC 207	FC 207	// Vibrator
"_352VI210"	FC 208	FC 208	// Vibrator
"_352VI211"	FC 209	FC 209	// Vibrator
"_352VI310"	FC 210	FC 210	// Vibrator
"_352VI311"	FC 211	FC 211	// Vibrator
"_EP100P1"	FC 212	FC 212	// EFilter Pole 1
"_EP100P2"	FC 213	FC 213	// EFilter Pole 2
"_SPARE_UNIMOTOR14"	FC 214	FC 214
"_SPARE_UNIMOTOR15"	FC 215	FC 215
"_SPARE_UNIMOTOR16"	FC 216	FC 216
"_SPARE_UNIMOTOR17"	FC 217	FC 217
"_SPARE_UNIMOTOR18"	FC 218	FC 218
"_SPARE_UNIMOTOR19"	FC 219	FC 219
"_SPARE_UNIMOTOR20"	FC 220	FC 220
"_411SD311"	FC 251	FC 251	// Gate Gypsum To Pneumatic Pump
"_411SD321"	FC 252	FC 252	// Gate Gypsum To Screw Conveyor
"_411SD331"	FC 253	FC 253	// Gate Weight 351BI100 Inlet
"_411SD332"	FC 254	FC 254	// Gate Weight 351BI200 Inlet
"_411SD333"	FC 255	FC 255	// Gate Weight 351BI300 Inlet
"_SPARE_VALVE06"	FC 256	FC 256
"_351SD141"	FC 257	FC 257	// Gate Boiler 1 Outlet
"_352SD120"	FC 258	FC 258	// Gate Weight 352BI100 Outlet
"_352SD121"	FC 259	FC 259	// Gate Weight 352BI100 Outlet
"_SPARE_VALVE10"	FC 260	FC 260
"_351SD241"	FC 261	FC 261	// Gate Boiler 2 Outlet
"_352SD220"	FC 262	FC 262	// Gate Weight 352BI200 Outlet
"_352SD221"	FC 263	FC 263	// Gate Weight 352BI200 Outlet
"_SPARE_VALVE14"	FC 264	FC 264
"_351SD341"	FC 265	FC 265	// Gate Boiler 3 Outlet
"_352SD320"	FC 266	FC 266	// Gate Weight 352BI300 Outlet
"_352SD321"	FC 267	FC 267	// Gate Weight 352BI300 Outlet
"_361SD170"	FC 268	FC 268	// Gate 371BI100 Inlet
"_361SD171"	FC 269	FC 269	// Gate 371BI200 Inlet
"_361SD172"	FC 270	FC 270	// Gate 371BI200 Inlet
"_361SD173"	FC 271	FC 271	// Gate 371BI300 Inlet
"_361SD174"	FC 272	FC 272	// Gate 371BI300 Inlet
"_361SD175"	FC 273	FC 273	// Gate 371BI400 Inlet
"_361SD176"	FC 274	FC 274	// Gate 371BI400 Inlet
"_361SD177"	FC 275	FC 275	// Gate 371BI500 Inlet
"_351BV031"	FC 276	FC 276	// Aqua to Boiler 1
"_351BV032"	FC 277	FC 277	// Aqua to Boiler 2
"_351BV033"	FC 278	FC 278	// Aqua to Boiler 3
"_351SD135"	FC 279	FC 279	// Gate Weight 351BI130
"_351SD235"	FC 280	FC 280	// Gate Weight 351BI230 Inlet
"_351SD335"	FC 281	FC 281	// Gate Weight 351BI300 Inlet
"_411BV151"	FC 282	FC 282	// Valve Separator Aspiration
"_SPARE_VALVE33"	FC 283	FC 283
"_351SD106"	FC 284	FC 284	// Gate Boiler 1 Outlet
"_351SD107"	FC 285	FC 285	// Gate Boiler 1 Outlet
"_351SD108"	FC 286	FC 286	// Gate Boiler 3 Outlet Hot Air
"_351SD109"	FC 287	FC 287	// Gate Hot Air To  Gypsum Line
"_SPARE_VALVE38"	FC 288	FC 288
"_SPARE_VALVE39"	FC 289	FC 289
"_SPARE_VALVE40"	FC 290	FC 290
"_SPARE_UMOTSC01"	FC 301	FC 301	// Chain Conveyor
"_143VF150"	FC 302	FC 302	// Vibrating Din
"_143BC160"	FC 303	FC 303	// Belt Conveyor
"_SPARE_UMOTSC04"	FC 304	FC 304	// Belt Conveyor
"_143RB250"	FC 305	FC 305	// Crusher
"_143BE300"	FC 306	FC 306	// Elevator
"_143FN122"	FC 307	FC 307	// Filter Fan
"_311RF200"	FC 308	FC 308	// Rotary Feeder
"_411FN101"	FC 309	FC 309	// Fan Crusher Drive Cooling
"_411RF201"	FC 310	FC 310	// Rotary Feeder
"_411RF304"	FC 311	FC 311	// Rotary Feeder
"_411SC322"	FC 312	FC 312	// Screw Conveyor
"_SPARE_UMOTSC13"	FC 313	FC 313
"_SPARE_UMOTSC14"	FC 314	FC 314
"_SPARE_UMOTSC15"	FC 315	FC 315
"_SPARE_UMOTSC16"	FC 316	FC 316
"_331RF301"	FC 317	FC 317	// Rotary Feeder
"_331RF302"	FC 318	FC 318	// Rotary Feeder
"_331RF303"	FC 319	FC 319	// Rotary Feeder
"_331SC351"	FC 320	FC 320	// Screw Conveyor
"_411RF314"	FC 321	FC 321	// Rotary Feeder
"_361SC150"	FC 322	FC 322	// Screw Conveyor
"_SPARE_UMOTSC23"	FC 323	FC 323
"_411PP312"	FC 324	FC 324	// Pneumatic Pump
"_SPARE_UMOTSC25"	FC 325	FC 325
"_SPARE_UMOTSC26"	FC 326	FC 326
"_351AG130"	FC 327	FC 327	// Mixer 1
"_351AG230"	FC 328	FC 328	// MIxer 2
"_351AG330"	FC 329	FC 329	// MIxer 3
"_361SC110"	FC 330	FC 330	// Screw Conveyor
"_361SC111"	FC 331	FC 331	// Screw Conveyor
"_361BE120"	FC 332	FC 332	// Elevator
"_361SC130"	FC 333	FC 333	// Screw Conveyor
"_SPARE_UMOTSC34"	FC 334	FC 334
"_361SC141"	FC 335	FC 335	// Screw Conveyor
"_SPARE_UMOTSC36"	FC 336	FC 336
"_361SC160"	FC 337	FC 337	// Screw Conveyor
"_341RF101_SPARE"	FC 338	FC 338	// Rotary Feeder
"_SPARE_UMOTSC39"	FC 339	FC 339
"_411FN200"	FC 340	FC 340	// Fan Hot Air To Crusher
"_351AG050"	FC 341	FC 341	// MIxer
"_351SP100"	FC 342	FC 342	// Pump
"_SPARE_UMOTSC43"	FC 343	FC 343
"_SPARE_UMOTSC44"	FC 344	FC 344
"_SPARE_UMOTSC45"	FC 345	FC 345
"_SPARE_UMOTSC46"	FC 346	FC 346
"_SPARE_UMOTSC47"	FC 347	FC 347
"_SPARE_UMOTSC48"	FC 348	FC 348
"_SPARE_UMOTSC49"	FC 349	FC 349
"_SPARE_UMOTSC50"	FC 350	FC 350
"_SPARE_UMOTSC51"	FC 351	FC 351
"_SPARE_UMOTSC52"	FC 352	FC 352
"_SPARE_UMOTSC53"	FC 353	FC 353
"_SPARE_UMOTSC54"	FC 354	FC 354
"_SPARE_UMOTSC55"	FC 355	FC 355
"_SPARE_UMOTSC56"	FC 356	FC 356
"_SPARE_UMOTSC57"	FC 357	FC 357
"_SPARE_UMOTSC58"	FC 358	FC 358
"_SPARE_UMOTSC59"	FC 359	FC 359
"_SPARE_UMOTSC60"	FC 360	FC 360
"_SPARE_UMOTSC61"	FC 361	FC 361
"_SPARE_UMOTSC62"	FC 362	FC 362
"_SPARE_UMOTSC63"	FC 363	FC 363
"_SPARE_UMOTSC64"	FC 364	FC 364
"_SPARE_UMOTSC65"	FC 365	FC 365
"_SPARE_UMOTSC66"	FC 366	FC 366
"_SPARE_UMOTSC67"	FC 367	FC 367
"_SPARE_UMOTSC68"	FC 368	FC 368
"_SPARE_UMOTSC69"	FC 369	FC 369
"_SPARE_UMOTSC70"	FC 370	FC 370
"_SPARE_UMOTSC71"	FC 371	FC 371
"_SPARE_UMOTSC72"	FC 372	FC 372
"_SPARE_UMOTSC73"	FC 373	FC 373
"_SPARE_UMOTSC74"	FC 374	FC 374
"_SPARE_UMOTSC75"	FC 375	FC 375
"_SPARE_UMOTSC76"	FC 376	FC 376
"_SPARE_UMOTSC77"	FC 377	FC 377
"_SPARE_UMOTSC78"	FC 378	FC 378
"_SPARE_UMOTSC79"	FC 379	FC 379
"_SPARE_UMOTSC80"	FC 380	FC 380
"_SPARE_UMOTSC81"	FC 381	FC 381
"_SPARE_UMOTSC82"	FC 382	FC 382
"_SPARE_UMOTSC83"	FC 383	FC 383
"_SPARE_UMOTSC84"	FC 384	FC 384
"_SPARE_UMOTSC85"	FC 385	FC 385
"_SPARE_UMOTSC86"	FC 386	FC 386
"_SPARE_UMOTSC87"	FC 387	FC 387
"_SPARE_UMOTSC88"	FC 388	FC 388
"_SPARE_UMOTSC89"	FC 389	FC 389
"_SPARE_UMOTSC90"	FC 390	FC 390
"_SPARE_UMOTSC91"	FC 391	FC 391
"_SPARE_UMOTSC92"	FC 392	FC 392
"_SPARE_UMOTSC93"	FC 393	FC 393
"_SPARE_UMOTSC94"	FC 394	FC 394
"_SPARE_UMOTSC95"	FC 395	FC 395
"_SPARE_UMOTSC96"	FC 396	FC 396
"_SPARE_UMOTSC97"	FC 397	FC 397
"_SPARE_UMOTSC98"	FC 398	FC 398
"_SPARE_UMOTSC99"	FC 399	FC 399
"_331LD391"	FC 401	FC 401	// Gate Filter Fan
"_331LD392"	FC 402	FC 402	// Gate Filter Fan
"_SPARE_AGATESC03"	FC 403	FC 403
"_SPARE_AGATESC04"	FC 404	FC 404
"_SPARE_AGATESC05"	FC 405	FC 405
"_SPARE_AGATESC06"	FC 406	FC 406
"_SPARE_AGATESC07"	FC 407	FC 407
"_SPARE_AGATESC08"	FC 408	FC 408
"_SPARE_AGATESC09"	FC 409	FC 409
"_SPARE_AGATESC10"	FC 410	FC 410
"_SPARE_GATESC01"	FC 451	FC 451
"_SPARE_GATESC02"	FC 452	FC 452
"_SPARE_GATESC03"	FC 453	FC 453
"_SPARE_GATESC04"	FC 454	FC 454
"_SPARE_GATESC05"	FC 455	FC 455
"_SPARE_GATESC06"	FC 456	FC 456
"_SPARE_GATESC07"	FC 457	FC 457
"_SPARE_GATESC08"	FC 458	FC 458
"_SPARE_GATESC09"	FC 459	FC 459
"_SPARE_GATESC10"	FC 460	FC 460
"_SPARE_BIMOTSC01"	FC 501	FC 501
"_SPARE_BIMOTSC02"	FC 502	FC 502
"_SPARE_BIMOTSC03"	FC 503	FC 503
"_SPARE_BIMOTSC04"	FC 504	FC 504
"_SPARE_BIMOTSC05"	FC 505	FC 505
"_SPARE_BIMOTSC06"	FC 506	FC 506
"_SPARE_BIMOTSC07"	FC 507	FC 507
"_SPARE_BIMOTSC08"	FC 508	FC 508
"_SPARE_BIMOTSC09"	FC 509	FC 509
"_SPARE_BIMOTSC10"	FC 510	FC 510
"_SPARE_BIMOTOR01"	FC 551	FC 551
"_SPARE_BIMOTOR02"	FC 552	FC 552
"_SPARE_BIMOTOR03"	FC 553	FC 553
"_SPARE_BIMOTOR04"	FC 554	FC 554
"_SPARE_BIMOTOR05"	FC 555	FC 555
"_SPARE_BIMOTOR06"	FC 556	FC 556
"_SPARE_BIMOTOR07"	FC 557	FC 557
"_SPARE_BIMOTOR08"	FC 558	FC 558
"_SPARE_BIMOTOR09"	FC 559	FC 559
"_SPARE_BIMOTOR10"	FC 560	FC 560
"_331FN401"	FC 601	FC 601	// Fan
"_411MD140"	FC 602	FC 602	// Crusher
"_311TF150"	FC 603	FC 603	// Rorary Table
"_411MD152"	FC 604	FC 604	// Separator
"_143BC200"	FC 605	FC 605	// Belt Conveyor
"_362SC140"	FC 606	FC 606	// Screw Conveyor
"_143CV100"	FC 607	FC 607	// Chain Conveyor
"_351SC120"	FC 608	FC 608	// Screw Conveyor
"_351SC220"	FC 609	FC 609	// Screw Conveyor
"_351SC320"	FC 610	FC 610	// Screw Conveyor
"_WF_GROUP"	FC 650	FC 650
"_SPARE_WF01"	FC 651	FC 651
"_SPARE_WF02"	FC 652	FC 652
"_SPARE_WF03"	FC 653	FC 653
"_SPARE_WF04"	FC 654	FC 654
"_SPARE_WF05"	FC 655	FC 655
"_SPARE_WF06"	FC 656	FC 656
"_SPARE_WF07"	FC 657	FC 657
"_SPARE_WF08"	FC 658	FC 658
"_SPARE_WF09"	FC 659	FC 659
"_SPARE_WF10"	FC 660	FC 660
"_SERVICE VALVE"	FC 700	FC 700
"_SERVICE UNIMOTOR"	FC 701	FC 701
"_SERVICE FC"	FC 702	FC 702
"_SERVICE POSITIONER"	FC 703	FC 703
"_SERVICE AI"	FC 704	FC 704
"_SERVICE GATE"	FC 705	FC 705
"_SERVICE AGATE"	FC 706	FC 706
"_SERVICE BIMOTOR"	FC 709	FC 709
"_SERVICE UMOT SC"	FC 710	FC 710
"_SERVICE BIMOT SC"	FC 711	FC 711
"_SERVICE GATE SC"	FC 712	FC 712
"_SERVICE AGATE SC"	FC 714	FC 714
"_SERVICE WF"	FC 715	FC 715
"_SPARE_GATE01"	FC 751	FC 751
"_SPARE_GATE02"	FC 752	FC 752
"_SPARE_GATE03"	FC 753	FC 753
"_SPARE_GATE04"	FC 754	FC 754
"_SPARE_GATE05"	FC 755	FC 755
"_SPARE_AGATE01"	FC 771	FC 771
"_SPARE_AGATE02"	FC 772	FC 772
"_SPARE_AGATE03"	FC 773	FC 773
"_SPARE_AGATE04"	FC 774	FC 774
"_SPARE_AGATE05"	FC 775	FC 775
"_BE300_LEVEL_MAX"	FC 801	FC 801	// Elevator Level Max Alarm
"_311BI100_LEVEL_H"	FC 802	FC 802	// 351BI100 Level Max Alarm
"_311BI100_LEVEL_L"	FC 803	FC 803	// 351BI100 Level Min Alarm
"_371BI100_LEVEL_H"	FC 804	FC 804	// 371BI100 Level Max Alarm
"_371BI100_LEVEL_L"	FC 805	FC 805	// 371BI100 Level Min Alarm
"_371BI200_LEVEL_H"	FC 806	FC 806	// 371BI200 Level Max Alarm
"_371BI200_LEVEL_L"	FC 807	FC 807	// 371BI200 Level Min Alarm
"_371BI300_LEVEL_H"	FC 808	FC 808	// 371BI300 Level Max Alarm
"_371BI300_LEVEL_L"	FC 809	FC 809	// 371BI300 Level Min Alarm
"_371BI400_LEVEL_H"	FC 810	FC 810	// 371BI400 Level Max Alarm
"_371BI400_LEVEL_L"	FC 811	FC 811	// 371BI400 Level Min Alarm
"_371BI500_LEVEL_H"	FC 812	FC 812	// 371BI500 Level Max Alarm
"_371BI500_LEVEL_L"	FC 813	FC 813	// 371BI500 Level Min Alarm
"_BE120_LEVEL_H"	FC 814	FC 814	// Elevator Level Max Alarm
"_341BI100_LEVEL_H"	FC 815	FC 815	// 341BI100 Level Max Alarm
"_341BI100_LEVEL_L"	FC 816	FC 816	// 341BI100 Level Min Alarm
"_331FN401_SELECTED"	FC 817	FC 817	// FN401 Selected
"_331FN402_SELECTED"	FC 818	FC 818	// FN402 Selected
"_441BI100_LEVEL_H"	FC 819	FC 819	// 441BI100 Level  Max Alarm
"_411BI100_LEVEL_L"	FC 820	FC 820	// 411BI100 Level Max Alarm
"_FA2_380V"	FC 821	FC 821	// Circuit switch 380 VAC - SITOP
"_FA22_220V"	FC 822	FC 822	// Circuit switch 220 VAC - Valve 1
"_K3UPS"	FC 823	FC 823	// Voltage before UPS - 220 VAC
"_FA20_220V"	FC 824	FC 824	// Circuit switch 220 VAC - Main voltage
"_FA3_24V"	FC 825	FC 825	// Circuit switch 24 VDC - MCC Main voltage
"_FA31_24V"	FC 826	FC 826	// Circuit switch 24 VDC - Main voltage
"_FA40_24V"	FC 827	FC 827	// Circuit switch 24 VDC - DO Moduls A7, A8
"_FA41_24V"	FC 828	FC 828	// Circuit switch 24 VDC - AI Modul A12
"_FA42_24V"	FC 829	FC 829	// Circuit switch 24 VDC - AI Modul A13
"_FA43_24V"	FC 830	FC 830	// Circuit switch 24 VDC - AI Modul A14
"_FA44_24V"	FC 831	FC 831	// Circuit switch 24 VDC - AI Modul A15
"_FA45_24V"	FC 832	FC 832	// Circuit switch 24 VDC - AI Modul A16
"_FA46_24V"	FC 833	FC 833	// Circuit switch 24 VDC - AI Modul A17
"_FA47_24V"	FC 834	FC 834	// Circuit switch 24 VDC - AO Modul A18
"_FA23_220V"	FC 835	FC 835	// Circuit switch 220 VAC - Valve 2
"_SR_OK"	FC 836	FC 836	// Safety Rellay OK
"_FA24_220V"	FC 837	FC 837	// Circuit switch 220 VAC - Light control and Horn
"_FA25_220V"	FC 838	FC 838	// Circuit switch 220 VAC - Level MIKMA
"_FA48_24V"	FC 839	FC 839	// Circuit switch 24 VDC - AI Modul A19
"_EF_DISCH_EN"	FC 840	FC 840	// EFilter Discharge Enable
"_EF_BIGBAG_FULL"	FC 841	FC 841	// EFilter Big Bag Full
"_SPARE_ALARM42"	FC 842	FC 842
"_SPARE_ALARM43"	FC 843	FC 843
"_SPARE_ALARM44"	FC 844	FC 844
"_SPARE_ALARM45"	FC 845	FC 845
"_SPARE_ALARM46"	FC 846	FC 846
"_SPARE_ALARM47"	FC 847	FC 847
"_SPARE_ALARM48"	FC 848	FC 848
"_SPARE_ALARM49"	FC 849	FC 849
"_SPARE_ALARM50"	FC 850	FC 850
"_SPARE_ALARM51"	FC 851	FC 851
"_SPARE_ALARM52"	FC 852	FC 852
"_SPARE_ALARM53"	FC 853	FC 853
"_SPARE_ALARM54"	FC 854	FC 854
"_SPARE_ALARM55"	FC 855	FC 855
"_SPARE_ALARM56"	FC 856	FC 856
"_SPARE_ALARM57"	FC 857	FC 857
"_SPARE_ALARM58"	FC 858	FC 858
"_SPARE_ALARM59"	FC 859	FC 859
"_SPARE_ALARM60"	FC 860	FC 860
"_SPARE_ALARM61"	FC 861	FC 861
"_SPARE_ALARM62"	FC 862	FC 862
"_SPARE_ALARM63"	FC 863	FC 863
"_SPARE_ALARM64"	FC 864	FC 864
"_SPARE_ALARM65"	FC 865	FC 865
"_SPARE_ALARM66"	FC 866	FC 866
"_SPARE_ALARM67"	FC 867	FC 867
"_SPARE_ALARM68"	FC 868	FC 868
"_SPARE_ALARM69"	FC 869	FC 869
"_SPARE_ALARM70"	FC 870	FC 870
"_SPARE_ALARM71"	FC 871	FC 871
"_SPARE_ALARM72"	FC 872	FC 872
"_SPARE_ALARM73"	FC 873	FC 873
"_SPARE_ALARM74"	FC 874	FC 874
"_SPARE_ALARM75"	FC 875	FC 875
"_SPARE_ALARM76"	FC 876	FC 876
"_SPARE_ALARM77"	FC 877	FC 877
"_SPARE_ALARM78"	FC 878	FC 878
"_SPARE_ALARM79"	FC 879	FC 879
"_SPARE_ALARM80"	FC 880	FC 880
"_SPARE_ALARM81"	FC 881	FC 881
"_SPARE_ALARM82"	FC 882	FC 882
"_SPARE_ALARM83"	FC 883	FC 883
"_SPARE_ALARM84"	FC 884	FC 884
"_SPARE_ALARM85"	FC 885	FC 885
"_SPARE_ALARM86"	FC 886	FC 886
"_SPARE_ALARM87"	FC 887	FC 887
"_SPARE_ALARM88"	FC 888	FC 888
"_SPARE_ALARM89"	FC 889	FC 889
"_SPARE_ALARM90"	FC 890	FC 890
"_SPARE_ALARM91"	FC 891	FC 891
"_SPARE_ALARM92"	FC 892	FC 892
"_SPARE_ALARM93"	FC 893	FC 893
"_SPARE_ALARM94"	FC 894	FC 894
"_SPARE_ALARM95"	FC 895	FC 895
"_SPARE_ALARM96"	FC 896	FC 896
"_SPARE_ALARM97"	FC 897	FC 897
"_SPARE_ALARM98"	FC 898	FC 898
"_SPARE_ALARM99"	FC 899	FC 899
"_FN401_SELECT"	FC 901	FC 901	// FN401 Select
"_FN402_SELECT"	FC 902	FC 902	// FN402 Select
"_NO_VIBDIN_SELECT"	FC 903	FC 903	// Without Vibrating Din Select
"_CRUSHER_LOAD_EN"	FC 904	FC 904	// Crusher Load Eanble
"_411PP312_ SELECT"	FC 905	FC 905	// Gypsum to Line 1
"_351BI100_SELECT"	FC 906	FC 906	// 351BI100 Load Enable
"_351BI200_SELECT"	FC 907	FC 907	// 351BI200 Load Enable
"_351BI300_SELECT"	FC 908	FC 908	// 351BI300 Load Enable
"_BOILER1_LOAD_EN"	FC 909	FC 909	// Boiler 1 Load Enable
"_BOILER2_LOAD_EN"	FC 910	FC 910	// Boiler 2 Load Enable
"_BOILER3_LOAD_EN"	FC 911	FC 911	// Boiler 3 Load Enable
"_352BI100_DISCH_EN"	FC 912	FC 912	// 352BI100 Discharge Enable
"_352BI200_DISCH_EN"	FC 913	FC 913	// 352BI200 Discharge Enable
"_352BI300_DISCH_EN"	FC 914	FC 914	// 352BI300 Discharge Enable
"_361SD170_SELECT"	FC 915	FC 915	// 361SD170 Select Load To Bin 500
"_361SD171_SELECT"	FC 916	FC 916	// 361SD170 Select Load To Bin 100
"_361SD172_SELECT"	FC 917	FC 917	// 361SD170 Select Load To Bin 100
"_361SD173_SELECT"	FC 918	FC 918	// 361SD170 Select Load To Bin 200
"_361SD174_SELECT"	FC 919	FC 919	// 361SD170 Select Load To Bin 200
"_361SD175_SELECT"	FC 920	FC 920	// 361SD170 Select Load To Bin 300
"_361SD176_SELECT"	FC 921	FC 921	// 361SD170 Select Load To Bin 300
"_361SD177_SELECT"	FC 922	FC 922	// 361SD170 Select Load To Bin 400
"_352SD121_SELECT"	FC 923	FC 923	// 352SD321_SELECT
"_352SD221_SELECT"	FC 924	FC 924	// _352SD221_SELECT
"_352SD321_SELECT"	FC 925	FC 925
"_REG_TBS_AUT_SELECT"	FC 926	FC 926
"_361SC111_SELECT"	FC 927	FC 927
"_REG_DiffP_ASep_SELECT"	FC 928	FC 928	// Regler DiffP After Separator Select
"_REG_Curr_MD140_SELECT"	FC 929	FC 929	// REgler Current Crusher MD140 Select
"_REG_DiffP_B3_SELECT"	FC 930	FC 930	// Regler Diff Pressure Boiler 3 Select
"_REG_DiffP_B1_SELECT"	FC 931	FC 931	// Regler Diff Pressure Boiler 1 Select
"_REG_DiffP_B2_SELECT"	FC 932	FC 932	// Regler Diff Pressure Boiler 2 Select
"_411SD301"	FC 1001	FC 1001	// Positioner Ciclone CN100 Outlet
"_411SD302"	FC 1002	FC 1002	// Positioner Cyclone 101 Outlet
"_351SD101"	FC 1003	FC 1003	// Positioner Boiler 1 Outlet
"_351SD102"	FC 1004	FC 1004	// Positioner Boiler 2 Outlet
"_351SD103"	FC 1005	FC 1005	// Positioner Boiler 3 Outlet
"_351SD104_"	FC 1006	FC 1006
"_351SD105_"	FC 1007	FC 1007
"I0.0"	I 0.0	BOOL	// FA2 - PVB 380VAC Sitop
"I0.1"	I 0.1	BOOL	// FA22 - PVB 220VAC VALVE 1
"I0.2"	I 0.2	BOOL	// K3UPS - POWER OK Before UPS
"I0.3"	I 0.3	BOOL	// FA20 - PVB 230VAC Оперативка
"I0.4"	I 0.4	BOOL	// FA3 - PVB 24VDC MCC Supply
"I0.5"	I 0.5	BOOL	// FA31 - PVB 24VDC Оперативка
"I0.6"	I 0.6	BOOL	// FA40 - PVB 24VDC DO MODUL A7, A8
"I0.7"	I 0.7	BOOL	// FA41 - PVB 24VDC AI MODUL A12
"I1.0"	I 1.0	BOOL	// FA42 - PVB 24VDC AI MODUL A13
"I1.1"	I 1.1	BOOL	// FA43 - PVB 24VDC AI MODUL A14
"I1.2"	I 1.2	BOOL	// FA44 - PVB 24VDC AI MODUL A15
"I1.3"	I 1.3	BOOL	// FA45 - PVB 24VDC AI MODUL A16
"I1.4"	I 1.4	BOOL	// FA46 - PVB 24VDC AI MODUL A17
"I1.5"	I 1.5	BOOL	// FA47 - PVB 24VDC AO MODUL A18
"I1.6"	I 1.6	BOOL	// FA23 - PVB 220VAC VALVE 2
"I1.7"	I 1.7	BOOL	// Safety Rellay OK
"I2.0"	I 2.0	BOOL	// FA23 - PVB 220VAC HORN and LIGHT CONTROL
"I2.1"	I 2.1	BOOL	// FA23 - PVB 220VAC LEVEL MIKMA
"I2.2"	I 2.2	BOOL	// FA48 - PVB 24VDC AI MODUL A19
"I2.3"	I 2.3	BOOL	// SPARE
"I2.4"	I 2.4	BOOL	// SPARE
"I2.5"	I 2.5	BOOL	// SPARE
"I2.6"	I 2.6	BOOL	// SPARE
"I2.7"	I 2.7	BOOL	// SPARE
"I3.0"	I 3.0	BOOL	// 143CV100D01 - Motion Detector
"I3.1"	I 3.1	BOOL	// 143BC160D01 - Motion Detector
"I3.2"	I 3.2	BOOL	// 143BC200D01 - Motion Detector
"I3.3"	I 3.3	BOOL	// 143BE300D01 - Motion Detector
"I3.4"	I 3.4	BOOL	// 143BE300L01 - Level Max
"I3.5"	I 3.5	BOOL	// 143BF120A01 - FAULT BF120
"I3.6"	I 3.6	BOOL	// 311BI100L01 - Level Min
"I3.7"	I 3.7	BOOL	// 311BI100L02 - Level Max
"I4.0"	I 4.0	BOOL	// 311RF200D01 - Motion Detector
"I4.1"	I 4.1	BOOL	// 411RF201D01 - Motion Detector
"I4.2"	I 4.2	BOOL	// 411RF304D01 - Motion Detector
"I4.3"	I 4.3	BOOL	// 411SC332D01 - Motion Detector
"I4.4"	I 4.4	BOOL
"I4.5"	I 4.5	BOOL
"I4.6"	I 4.6	BOOL
"I4.7"	I 4.7	BOOL
"I5.0"	I 5.0	BOOL	// 411SD311D01 - Limit Switch Open
"I5.1"	I 5.1	BOOL	// 411SD311D02 - Limit Switch Close
"I5.2"	I 5.2	BOOL	// 411SD321D01 - Limit Switch Open
"I5.3"	I 5.3	BOOL	// 411SD321D02 - Limit Switch Close
"I5.4"	I 5.4	BOOL	// 411SD331D01 - Limit Switch Open
"I5.5"	I 5.5	BOOL	// 411SD331D02 - Limit Switch Close
"I5.6"	I 5.6	BOOL	// 411SD332D01 - Limit Switch Open
"I5.7"	I 5.7	BOOL	// 411SD332D02 - Limit Switch Close
"I6.0"	I 6.0	BOOL	// 411SD333D01 - Limit Switch Open
"I6.1"	I 6.1	BOOL	// 411SD333D02 - Limit Switch Close
"I6.2"	I 6.2	BOOL
"I6.3"	I 6.3	BOOL
"I6.4"	I 6.4	BOOL
"I6.5"	I 6.5	BOOL
"I6.6"	I 6.6	BOOL
"I6.7"	I 6.7	BOOL
"I7.0"	I 7.0	BOOL
"I7.1"	I 7.1	BOOL
"I7.2"	I 7.2	BOOL	// 331RF301D01 - Motion Detector
"I7.3"	I 7.3	BOOL	// 331RF302D01 - Motion Detector
"I7.4"	I 7.4	BOOL	// 331RF303D01 - Motion Detector
"I7.5"	I 7.5	BOOL	// 331SC351D01 - Motion Detector
"I7.6"	I 7.6	BOOL	// 341SI100L01 - Level Min
"I7.7"	I 7.7	BOOL	// 341SI100L02 - Level Max
"I8.0"	I 8.0	BOOL	// 351SC120D01 - Motion Detector
"I8.1"	I 8.1	BOOL	// 351SC220D01 - Motion Detector
"I8.2"	I 8.2	BOOL	// 351SC320D01 - Motion Detector
"I8.3"	I 8.3	BOOL
"I8.4"	I 8.4	BOOL
"I8.5"	I 8.5	BOOL	// 351SD141D01 - Limit Switch Open
"I8.6"	I 8.6	BOOL	// 351SD141D02 - Limit Switch Close
"I8.7"	I 8.7	BOOL	// 352SD120D01 - Limit Switch Open
"I9.0"	I 9.0	BOOL	// 352SD120D02 - Limit Switch Close
"I9.1"	I 9.1	BOOL	// 352SD121D01 - Limit Switch Open
"I9.2"	I 9.2	BOOL	// 352SD121D02 - Limit Switch Close
"I9.3"	I 9.3	BOOL
"I9.4"	I 9.4	BOOL
"I9.5"	I 9.5	BOOL	// 351SD241D01 - Limit Switch Open
"I9.6"	I 9.6	BOOL	// 351SD241D02 - Limit Switch Close
"I9.7"	I 9.7	BOOL	// 352SD220D01 - Limit Switch Open
"I10.0"	I 10.0	BOOL	// 352SD220D02 - Limit Switch Close
"I10.1"	I 10.1	BOOL	// 352SD221D01 - Limit Switch Open
"I10.2"	I 10.2	BOOL	// 352SD221D02 - Limit Switch Close
"I10.3"	I 10.3	BOOL	// 361SC160D01 - Motion Detector
"I10.4"	I 10.4	BOOL
"I10.5"	I 10.5	BOOL	// 351SD341D01 - Limit Switch Open
"I10.6"	I 10.6	BOOL	// 351SD341D02 - Limit Switch Close
"I10.7"	I 10.7	BOOL	// 352SD320D01 - Limit Switch Open
"I11.0"	I 11.0	BOOL	// 352SD320D02 - Limit Switch Close
"I11.1"	I 11.1	BOOL	// 352SD321D01 - Limit Switch Open
"I11.2"	I 11.2	BOOL	// 352SD321D02 - Limit Switch Close
"I11.3"	I 11.3	BOOL	// 361SC110D01 - Motion Detector
"I11.4"	I 11.4	BOOL	// 361SC111D01 - Motion Detector
"I11.5"	I 11.5	BOOL	// 361BE120D01 - Motion Detector
"I11.6"	I 11.6	BOOL	// 361BE120L01 - Level Max
"I11.7"	I 11.7	BOOL	// 361SC130D01 - Motion Detector
"I12.0"	I 12.0	BOOL	// 361SC140D01 - Motion Detector
"I12.1"	I 12.1	BOOL	// 361SC141D01 - Motion Detector
"I12.2"	I 12.2	BOOL	// 361SC150D01 - Motion Detector
"I12.3"	I 12.3	BOOL	// 361SD170D01 - Limit Switch Open
"I12.4"	I 12.4	BOOL	// 361SD170D02 - Limit Switch Close
"I12.5"	I 12.5	BOOL	// 361SD171D01 - Limit Switch Open
"I12.6"	I 12.6	BOOL	// 361SD171D02 - Limit Switch Close
"I12.7"	I 12.7	BOOL	// 361SD172D01 - Limit Switch Open
"I13.0"	I 13.0	BOOL	// 361SD172D02 - Limit Switch Close
"I13.1"	I 13.1	BOOL	// 361SD173D01 - Limit Switch Open
"I13.2"	I 13.2	BOOL	// 361SD173D02 - Limit Switch Close
"I13.3"	I 13.3	BOOL	// 361SD174D01 - Limit Switch Open
"I13.4"	I 13.4	BOOL	// 361SD174D02 - Limit Switch Close
"I13.5"	I 13.5	BOOL	// 361SD175D01 - Limit Switch Open
"I13.6"	I 13.6	BOOL	// 361SD175D02 - Limit Switch Close
"I13.7"	I 13.7	BOOL	// 361SD176D01 - Limit Switch Open
"I14.0"	I 14.0	BOOL	// 361SD176D02 - Limit Switch Close
"I14.1"	I 14.1	BOOL	// 361SD177D01 - Limit Switch Open
"I14.2"	I 14.2	BOOL	// 361SD177D02 - Limit Switch Close
"I14.3"	I 14.3	BOOL
"I14.4"	I 14.4	BOOL
"I14.5"	I 14.5	BOOL
"I14.6"	I 14.6	BOOL
"I14.7"	I 14.7	BOOL	// 351SD106D01 - Limit Switch Open
"I15.0"	I 15.0	BOOL	// 351SD106D02 - Limit Switch Close
"I15.1"	I 15.1	BOOL	// 351SD107D01 - Limit Switch Open
"I15.2"	I 15.2	BOOL	// 351SD107D02 - Limit Switch Close
"I15.3"	I 15.3	BOOL	// 351SD108D01 - Limit Switch Open
"I15.4"	I 15.4	BOOL	// 351SD108D02 - Limit Switch Close
"I15.5"	I 15.5	BOOL	// 351SD109D01 - Limit Switch Open
"I15.6"	I 15.6	BOOL	// 351SD109D02 - Limit Switch Close
"I15.7"	I 15.7	BOOL
"I16.0"	I 16.0	BOOL	// 351VI110FA1 - PVB
"I16.1"	I 16.1	BOOL	// 351VI110KM1 - Contactor
"I16.2"	I 16.2	BOOL	// 351VI210FA1 - PVB
"I16.3"	I 16.3	BOOL	// 351VI210KM1 - Contactor
"I16.4"	I 16.4	BOOL	// 351VI310FA1 - PVB
"I16.5"	I 16.5	BOOL	// 351VI310KM1 - Contactor
"I16.6"	I 16.6	BOOL	// 352VI110FA1 - PVB
"i16.7"	I 16.7	BOOL	// 352VI110KM - Contactor
"I17.0"	I 17.0	BOOL	// 352VI111FA1 - PVB
"I17.1"	I 17.1	BOOL	// 352VI111KM1 - Contactor
"I17.2"	I 17.2	BOOL	// 352VI210FA1 - PVB
"I17.3"	I 17.3	BOOL	// 352VI210KM1 - Contactor
"117.4"	I 17.4	BOOL	// 352VI211FA1 - PVB
"I17.5"	I 17.5	BOOL	// 352VI211KM1 - Contactor
"I17.6"	I 17.6	BOOL	// 352VI310FA1 - PVB
"I17.7"	I 17.7	BOOL	// 352VI310KM1 - Contactor
"I18.0"	I 18.0	BOOL	// 352VI311FA1 - PVB
"I18.1"	I 18.1	BOOL	// 352VI311KM1 - Contactor
"I18.2"	I 18.2	BOOL	// FA10 - PVB - SPARE
"I18.3"	I 18.3	BOOL	// KM10 - Contactor - SPARE
"I18.4"	I 18.4	BOOL	// 361SC110_RUN
"I18.5"	I 18.5	BOOL	// 361SC111_RUN
"I18.6"	I 18.6	BOOL	// SPARE MCC
"I18.7"	I 18.7	BOOL	// SPARE MCC
"I20.0"	I 20.0	BOOL	// 351SD135D01 - Limit Switch Open
"I20.1"	I 20.1	BOOL	// 351SD135D02 - Limit Switch Close
"I20.2"	I 20.2	BOOL	// 351SD235D01 - Limit Switch Open
"I20.3"	I 20.3	BOOL	// 351SD235D02 - Limit Switch Close
"I20.4"	I 20.4	BOOL	// 351SD335D01 - Limit Switch Open
"I20.5"	I 20.5	BOOL	// 351SD335D02 - Limit Switch Close
"I20.6"	I 20.6	BOOL	// 351BI100D01L41 - Level MIKMA
"I20.7"	I 20.7	BOOL	// 351BI200D01L41 - Level MIKMA
"I21.0"	I 21.0	BOOL	// 351BI300D01L41 - Level MIKMA
"I21.1"	I 21.1	BOOL	// 351BI400D01L41 - Level MIKMA
"I21.2"	I 21.2	BOOL	// 351BI500D01L41 - Level MIKMA
"I21.3"	I 21.3	BOOL	// 441BI100D01L41 - High Level MIKMA
"I21.4"	I 21.4	BOOL	// 441BI100D02L41 - Low Level MIKMA
"I21.5"	I 21.5	BOOL	// SPARE Level MIKMA
"I21.6"	I 21.6	BOOL	// EF Discharge Stop Button
"I21.7"	I 21.7	BOOL	// EFilter BigBag Full
"I22.0"	I 22.0	BOOL	// SPARE PLC
"I22.1"	I 22.1	BOOL	// SPARE PLC
"I22.2"	I 22.2	BOOL	// SPARE PLC
"I22.3"	I 22.3	BOOL	// SPARE PLC
"I22.4"	I 22.4	BOOL	// SPARE PLC
"i22.5"	I 22.5	BOOL	// SPARE PLC
"I22.6"	I 22.6	BOOL	// SPARE PLC
"I22.7"	I 22.7	BOOL	// SPARE PLC
"I23.0"	I 23.0	BOOL	// TS1 Department Stop 1
"I23.1"	I 23.1	BOOL	// TS2 Department Stop 2
"I23.2"	I 23.2	BOOL	// TS3 Department Stop 3
"I23.3"	I 23.3	BOOL	// TS4 Department Stop 4
"I23.4"	I 23.4	BOOL	// TS5 Department Stop 5
"I23.5"	I 23.5	BOOL	// TS6 Department Stop 6
"I23.6"	I 23.6	BOOL	// TS7 Department Stop 7
"I23.7"	I 23.7	BOOL	// TS8 Department Stop 8
"P1_Status"	I 201.0	BOOL	// Status VAP, 1 - ON, 0 - OFF
"P1_Alarm"	I 201.1	BOOL	// Alarm, 1 - Alarm
"P1_Low_Voltage"	I 204.0	BOOL	// Alarm - Low voltage more than 30 s, 1 - Alarm
"P1_High_Voltage"	I 204.1	BOOL	// Alarm - High voltage more than 1 s, 1 - Alarm
"P1_Sinhronization"	I 204.2	BOOL	// Alarm - NO sinhronization, 1 - Alarm
"P1_High_Oil_Pressure_VAP"	I 205.0	BOOL	// Alarm - High oil pressure VAP, 1 - Alarm
"P1_High_Temperature_VAP"	I 205.1	BOOL	// Alarm - High temperature VAP, 1 - Alarm
"P1_Low_Oil_Level_VAP"	I 205.2	BOOL	// Alarm - Low oil level VAP, 1 - Alarm
"P1_VAP_Grounded"	I 205.3	BOOL	// Alarm - VAP Grounded, 1 - Alarm
"P1_High_Temp_Tiristor"	I 205.4	BOOL	// Alarm - High temperature tiristor, 1 - Alarm
"P1_Main_Switch"	I 205.5	BOOL	// Alarm - Main switch, 1 - Alarm
"P1_VAP_Blocked"	I 205.6	BOOL	// Alarm - VAP blocked, 1 - Alarm
"P1_Main_Conntactor"	I 205.7	BOOL	// Alarm - Main conntactor, 1 - Alarm
"P1_Rapping_Motor1"	I 208.0	BOOL	// System rappind motor 1 ON, 1 - ON, 0 - OFF
"P1_Rapping_Motor2"	I 208.1	BOOL	// System rappind motor 2 ON, 1 - ON, 0 - OFF
"P1_Rapping_Motor3"	I 208.2	BOOL	// System rappind motor 3 ON, 1 - ON, 0 - OFF
"P1_Rapping_Motor1_Alarm"	I 208.3	BOOL	// System rappind motor 1 Alarm, 1 - Alarm
"P1_Rapping_Motor2_Alarm"	I 208.4	BOOL	// System rappind motor 2 Alarm, 1 - Alarm
"P1_Rapping_Motor3_Alarm"	I 208.5	BOOL	// System rappind motor 3 Alarm, 1 - Alarm
"P1_Rapping_ON"	I 209.0	BOOL	// System rappind ON, 1 - ON, 0 - OFF
"P1_Rapping_Alarm"	I 209.1	BOOL	// System rappind alarm, 1 - Alarm
"P1_Rapping_Status"	I 209.2	BOOL	// System rappind status, 1 - External, 0 - Timer
"P1_Rapping_Parametr"	I 209.3	BOOL	// System rappind parametr, 1 - Main, 0 - Extended
"P1_Rapp_Mot1_Alarm_Loc"	I 212.0	BOOL	// System rappind motor 1 Local switch Alarm, 1 - Alarm
"P1_Rapp_Mot2_Alarm_Loc"	I 212.1	BOOL	// System rappind motor 2 Local switch Alarm, 1 - Alarm
"P1_Rapp_Mot3_Alarm_Loc"	I 212.2	BOOL	// System rappind motor 3 Local switch Alarm, 1 - Alarm
"P1_Rapp_Mot1_Alarm_Con"	I 213.0	BOOL	// System rappind motor 1 Contactor Alarm, 1 - Alarm
"P1_Rapp_Mot2_Alarm_Con"	I 213.1	BOOL	// System rappind motor 2 Contactor Alarm, 1 - Alarm
"P1_Rapp_Mot3_Alarm_Con"	I 213.2	BOOL	// System rappind motor 3 Contactor Alarm, 1 - Alarm
"P1_Rapp_Mot1_Alarm_Switc"	I 213.3	BOOL	// System rappind motor 1 Main switch Alarm, 1 - Alarm
"P1_Rapp_Mot2_Alarm_Switc"	I 213.4	BOOL	// System rappind motor 2 Main switch Alarm, 1 - Alarm
"P1_Rapp_Mot3_Alarm_Switc"	I 213.5	BOOL	// System rappind motor 3 Main switch Alarm, 1 - Alarm
"P2_Status"	I 233.0	BOOL	// Status VAP, 1 - ON, 0 - OFF
"P2_Alarm"	I 233.1	BOOL	// Alarm, 1 - Alarm
"P2_Low_Voltage"	I 236.0	BOOL	// Alarm - Low voltage more than 30 s, 1 - Alarm
"P2_High_Voltage"	I 236.1	BOOL	// Alarm - High voltage more than 1 s, 1 - Alarm
"P2_Sinhronization"	I 236.2	BOOL	// Alarm - NO sinhronization, 1 - Alarm
"P2_High_Oil_Pressure_VAP"	I 237.0	BOOL	// Alarm - High oil pressure VAP, 1 - Alarm
"P2_High_Temperature_VAP"	I 237.1	BOOL	// Alarm - High temperature VAP, 1 - Alarm
"P2_Low_Oil_Level_VAP"	I 237.2	BOOL	// Alarm - Low oil level VAP, 1 - Alarm
"P2_VAP_Grounded"	I 237.3	BOOL	// Alarm - VAP Grounded, 1 - Alarm
"P2_High_Temp_Tiristor"	I 237.4	BOOL	// Alarm - High temperature tiristor, 1 - Alarm
"P2_Main_Switch"	I 237.5	BOOL	// Alarm - Main switch, 1 - Alarm
"P2_VAP_Blocked"	I 237.6	BOOL	// Alarm - VAP blocked, 1 - Alarm
"P2_Main_Conntactor"	I 237.7	BOOL	// Alarm - Main conntactor, 1 - Alarm
"P2_Rapping_Motor1"	I 240.0	BOOL	// System rappind motor 1 ON, 1 - ON, 0 - OFF
"P2_Rapping_Motor2"	I 240.1	BOOL	// System rappind motor 2 ON, 1 - ON, 0 - OFF
"P2_Rapping_Motor3"	I 240.2	BOOL	// System rappind motor 3 ON, 1 - ON, 0 - OFF
"P2_Rapping_Motor1_Alarm"	I 240.3	BOOL	// System rappind motor 1 Alarm, 1 - Alarm
"P2_Rapping_Motor2_Alarm"	I 240.4	BOOL	// System rappind motor 2 Alarm, 1 - Alarm
"P2_Rapping_Motor3_Alarm"	I 240.5	BOOL	// System rappind motor 3 Alarm, 1 - Alarm
"P2_Rapping_ON"	I 241.0	BOOL	// System rappind ON, 1 - ON, 0 - OFF
"P2_Rapping_Alarm"	I 241.1	BOOL	// System rappind alarm, 1 - Alarm
"P2_Rapping_Status"	I 241.2	BOOL	// System rappind status, 1 - External, 0 - Timer
"P2_Rapping_Parametr"	I 241.3	BOOL	// System rappind parametr, 1 - Main, 0 - Extended
"P2_Rapp_Mot1_Alarm_Loc"	I 244.0	BOOL	// System rappind motor 1 Local switch Alarm, 1 - Alarm
"P2_Rapp_Mot2_Alarm_Loc"	I 244.1	BOOL	// System rappind motor 2 Local switch Alarm, 1 - Alarm
"P2_Rapp_Mot3_Alarm_Loc"	I 244.2	BOOL	// System rappind motor 3 Local switch Alarm, 1 - Alarm
"P2_Rapp_Mot1_Alarm_Con"	I 245.0	BOOL	// System rappind motor 1 Contactor Alarm, 1 - Alarm
"P2_Rapp_Mot2_Alarm_Con"	I 245.1	BOOL	// System rappind motor 2 Contactor Alarm, 1 - Alarm
"P2_Rapp_Mot3_Alarm_Con"	I 245.2	BOOL	// System rappind motor 3 Contactor Alarm, 1 - Alarm
"P2_Rapp_Mot1_Alarm_Switc"	I 245.3	BOOL	// System rappind motor 1 Main switch Alarm, 1 - Alarm
"P2_Rapp_Mot2_Alarm_Switc"	I 245.4	BOOL	// System rappind motor 2 Main switch Alarm, 1 - Alarm
"P2_Rapp_Mot3_Alarm_Switc"	I 245.5	BOOL	// System rappind motor 3 Main switch Alarm, 1 - Alarm
"IW64"	IW 64	INT	// 411DC100N01T01 - Температура перед дробаркою
"IW66"	IW 66	INT	// 411DC100N02P01 - Тиск перед дробаркою
"IW68"	IW 68	INT	// 411DC100N03T02 - Температура після дробарки
"IW70"	IW 70	INT	// 411DC100N04P02 - Тиск після дробарки
"IW72"	IW 72	INT	// 351BR300N06T04 - Температура гарячого повітря на бинтову лінію
"IW74"	IW 74	INT	// 351BR300N07P03 - Тиск гарячого повітря на бинтову лінію
"IW76"	IW 76	INT	// 351BI100N01T01 - Температура в бункері
"IW78"	IW 78	INT	// 351BI200N01T01 - Температура в бунекрі
"IW80"	IW 80	INT	// 351BI300N01T01 - Температура в бунекр
"IW82"	IW 82	INT	// 351BR100N01T01 - Температура в казані 1 верх
"IW84"	IW 84	INT	// 351BR100N02T02 - Температура в казані 1 низ
"IW86"	IW 86	INT	// 351BR100N03P01 - Розрідження в казані 1 низ
"IW88"	IW 88	INT	// 351BR200N01T01 - Температура в казані 2 верх
"IW90"	IW 90	INT	// 351BR200N02T02 - Температура в казані 2 низ
"IW92"	IW 92	INT	// 351BR200N03P01 - Розрідження в казані 2 низ
"IW94"	IW 94	INT	// 351BR300N02T01 - Температура в казані 3 верх
"IW96"	IW 96	INT	// 351BR300N02T02 - Температура в казані 3 низ
"IW98"	IW 98	INT	// 351BR300N03P01 - Розрідження в казані 3 низ
"IW100"	IW 100	INT	// 351BI100N02W01 - Вага бункера
"IW102"	IW 102	INT	// 351BI200N02W01 - Вага бункера
"IW104"	IW 104	INT	// 351BI300N02W01 - Вага бункера
"IW106"	IW 106	INT	// 352BI100N01W01 - Вага бункера
"IW108"	IW 108	INT	// 352BI200N01W01 - Вага бункера
"IW110"	IW 110	INT	// 352BI300N01W01 - Вага бункера
"IW112"	IW 112	INT	// 351BI130N01W01 - Вага бункера
"IW114"	IW 114	INT	// 351BI230N01W01 - Вага бункера
"IW116"	IW 116	INT	// 351BI330N01W01 - Вага бункера
"IW118"	IW 118	INT	// 331EP100N01P01 - Розрідження перед електрофільтром
"IW120"	IW 120	INT	// 331EP100N02T01  - Температура перед електрофільтром
"IW122"	IW 122	INT	// 331EP100N03T02 - Температура після електрофільтра
"IW124"	IW 124	INT	// 331EP100N04P02 - Розрідження після електрофільтра
"IW126"	IW 126	INT	// 411SD301Z01 - Положення засувки
"IW128"	IW 128	INT	// 411SD302Z01 - Положення засувки
"IW130"	IW 130	INT	// 411CN101N01P01 - Розрідження перед циклоном CN101
"IW132"	IW 132	INT	// 411CN101N02T01 - Темпереатура перед циклоном CN101
"IW134"	IW 134	INT	// 411CN101N03P02 - Розрідження після циклона CN101
"IW136"	IW 136	INT	// 411CN101N04T02 - Температура після циклона CN101
"IW138"	IW 138	INT	// 411CN103N01P01 - Розрідження після циклона CN103
"IW140"	IW 140	INT	// 411CN103N02T01 - Температура піля циклона CN103
"IW142"	IW 142	INT	// 351BR100N04T03 - Температура в топці казана 1
"IW144"	IW 144	INT	// 351BR100N05P02 - Розрідження в топці казана 1
"IW146"	IW 146	INT	// 351BR200N04T03 - Температура в топці казана 2
"IW148"	IW 148	INT	// 351BR200N05P02 - Розрідження в топці казана 2
"IW150"	IW 150	INT	// 351BR300N04T03 - Температура в топці казана 3
"IW152"	IW 152	INT	// 351BR300N05P02 - Розрідження в топці казана 3
"IW154"	IW 154	INT	// 351BR100N06T04 - Температура гарячих газів з котла 1 в дробарку
"IW156"	IW 156	INT	// 351BR200N06T04 - Температура гарячих газів з котла 2 в дробарку
"IW158"	IW 158	INT	// 351BR300N06T04 - Температура гарячих газів з котла 3 в дробарку
"IW160"	IW 160	INT	// 411SR150N03T02 - Температура перед сепаратором (підшипника)
"IW162"	IW 162	INT	// 351SD101Z01 - Положення засувки
"IW164"	IW 164	INT	// 351SD102Z01 - Положення засувки
"IW166"	IW 166	INT	// 351SD103Z01 - Положення засувки
"IW168"	IW 168	INT	// 351SD104Z01 - Положення засувки
"IW170"	IW 170	INT	// 351SD105Z01 - Положення засувки
"IW172"	IW 172	INT	// 100CP100N01P01 Pressure After Compressor
"IW174"	IW 174	INT
"IW176"	IW 176	INT
"IW178"	IW 178	INT
"IW180"	IW 180	INT
"IW182"	IW 182	INT
"IW184"	IW 184	INT
"IW186"	IW 186	INT
"IW188"	IW 188	INT
"IW190"	IW 190	INT
"P1_Main_Current"	IW 216	WORD	// Main Current I, A (0...500)
"P1_Aver_Current IDC"	IW 220	WORD	// Averege Current IDC, mA (0...2000)
"P1_Voltage"	IW 224	WORD	// Averege Voltage UDC*10, kV (0...2000)
"P2_Main_Current"	IW 248	WORD	// Main Current I, A (0...500)
"P2_Aver_Current IDC"	IW 252	WORD	// Averege Current IDC, mA (0...2000)
"P2_Voltage"	IW 256	WORD	// Averege Voltage UDC*10, kV (0...2000)
"0"	M 0.0	BOOL	// LOG 0
"1"	M 0.1	BOOL	// LOG 1
"M0.4"	M 0.4	BOOL	// First Scan
"SIM_ON"	M 0.5	BOOL	// Simulation ON/OFF
"M0.6"	M 0.6	BOOL	// One scan puls period 1 min
"Clock_1s"	M 1.0	BOOL	// Clock memory period  0.1 s
"Clock_2s"	M 1.1	BOOL	// Clock memory period  0.2 s
"Clock_4s"	M 1.2	BOOL	// Clock memory period  0.4 s
"Clock_5s"	M 1.3	BOOL	// Clock memory period  0.5 s
"Clock_8s"	M 1.4	BOOL	// Clock memory period  0.8 s
"Clock1s"	M 1.5	BOOL	// Clock memory period  1 s
"Clock1_6s"	M 1.6	BOOL	// Clock memory period  1.6 s
"Clock2s"	M 1.7	BOOL	// Clock memory period  2 s
"puls_1s"	M 2.0	BOOL	// One scan puls period 0.1 s
"puls_2s"	M 2.1	BOOL	// One scan puls period 0.2 s
"puls_4s"	M 2.2	BOOL	// One scan puls period 0.4 s
"puls_5s"	M 2.3	BOOL	// One scan puls period 0.5 s
"puls_8s"	M 2.4	BOOL	// One scan puls period 0.8 s
"puls1s"	M 2.5	BOOL	// One scan puls period 1 s
"puls1_6s"	M 2.6	BOOL	// One scan puls period 1.6 s
"puls2s"	M 2.7	BOOL	// One scan puls period 2 s
"Pclock_1s"	M 3.0	BOOL	// Positive edge clock 0.1 s
"Pclock_2s"	M 3.1	BOOL	// Positive edge clock 0.1 s
"Pclock_4s"	M 3.2	BOOL	// Positive edge clock 0.4 s
"Pclock_5s"	M 3.3	BOOL	// Positive edge clock 0.5 s
"Pclock_8s"	M 3.4	BOOL	// Positive edge clock 0.8 s
"Pclock1s"	M 3.5	BOOL	// Positive edge clock 1 s
"Pclock1_6s"	M 3.6	BOOL	// Positive edge clock 1.6 s
"Pclock2s"	M 3.7	BOOL	// Positive edge clock 2 s
"HSTP"	M 20.0	BOOL	// Hard Stop
"M61.0"	M 61.0	BOOL	// Load To 351BI100 Enable
"M61.1"	M 61.1	BOOL	// Discharge From 351BI10 Enable
"M61.2"	M 61.2	BOOL	// End Feeding From 351BI100
"M62.0"	M 62.0	BOOL	// Load to 351BI200 Enable
"M62.1"	M 62.1	BOOL	// Discharge form 351BI200 Enable
"M62.2"	M 62.2	BOOL	// End Feeding From 351BI200
"M63.0"	M 63.0	BOOL	// Load to 351BI300 Enable
"M63.1"	M 63.1	BOOL	// Discharge from 351BI300 Enable
"M63.2"	M 63.2	BOOL	// End Feeding From 351BI300
"M64.0"	M 64.0	BOOL	// Enable Load to 352BI100
"M64.1"	M 64.1	BOOL	// Discharge enable from 352BI100
"M64.2"	M 64.2	BOOL	// End Feeding From 352BI100
"M67.0"	M 67.0	BOOL	// Load Enable To BI130
"M67.1"	M 67.1	BOOL	// Discharge Enable From Bi130
"M67.2"	M 67.2	BOOL	// End Feeding  from BI130
"M68.0"	M 68.0	BOOL	// Enable Load to Weight 351BI230
"M68.1"	M 68.1	BOOL	// Discharge Enable From 351BI230
"M68.2"	M 68.2	BOOL	// End Feeding From BI230
"M69.0"	M 69.0	BOOL	// Enable Load to BI330
"M69.1"	M 69.1	BOOL	// Enable Discharge from BI330
"M69.2"	M 69.2	BOOL	// End Feeding Fom BI330
"M70.0"	M 70.0	BOOL	// Enable Load To Boiler 1
"M70.1"	M 70.1	BOOL	// Discharge From Boiler 1 Enable
"M70.2"	M 70.2	BOOL	// End Feeding From Boiler 1
"M71.0"	M 71.0	BOOL	// Load To Boiler 2 Enable
"M71.1"	M 71.1	BOOL	// Discharge From Boiler 2 Enable
"M71.2"	M 71.2	BOOL	// End Feeding From Boiler 2
"M72.0"	M 72.0	BOOL	// Load Enable To Boiler 3
"M72.1"	M 72.1	BOOL	// Discharge Enable From Boiler 3
"M72.2"	M 72.2	BOOL	// End Feeding From Boiler 3
"411MD150OVC"	M 80.0	BOOL	// Main drive over current
"M177.0"	M 177.0	BOOL	// BE120 current OK
"M203.0"	M 203.0	BOOL	// FP 351VI110 ON
"M203.1"	M 203.1	BOOL	// FP 351VI110 OFF
"M204.0"	M 204.0	BOOL	// FP 351VI210 ON
"M204.1"	M 204.1	BOOL	// FP 351VI210 OFF
"M205.0"	M 205.0	BOOL	// FP 351VI310 ON
"M205.1"	M 205.1	BOOL	// FP 351VI310 OFF
"M206.0"	M 206.0	BOOL	// FP 352VI110 ON
"M206.1"	M 206.1	BOOL	// FP 352VI110 OFF
"M207.0"	M 207.0	BOOL	// FP 352VI111 ON
"M207.1"	M 207.1	BOOL	// FP 352VI11 OFF
"M208.0"	M 208.0	BOOL	// FP 352VI210 ON
"M208.1"	M 208.1	BOOL	// FP 352VI210 OFF
"M209.0"	M 209.0	BOOL	// FP 352VI211 ON
"M209.1"	M 209.1	BOOL	// FP 352VI211 OFF
"M210.0"	M 210.0	BOOL	// FP 352VI310 ON
"M210.1"	M 210.1	BOOL	// FP 352VI310 OFF
"M211.0"	M 211.0	BOOL	// FP 352VI311 ON
"M211.1"	M 211.1	BOOL	// FP 352VI311 OFF
"M279.0"	M 279.0	BOOL	// Open SD135
"M280.0"	M 280.0	BOOL	// Open SD235
"M281.0"	M 281.0	BOOL	// Open SD335
"M282.0"	M 282.0	BOOL	// BV151  Open
"M401.0"	M 401.0	BOOL	// Gate LD351 Clased
"M402.0"	M 402.0	BOOL	// Gate LD392 Closed
"M604.0"	M 604.0	BOOL	// Separtor ON
"CYC_INT2"	OB 32	OB 32	// Cyclic Interrupt 2
"CYC_INT3"	OB 33	OB 33	// Cyclic Interrupt 3
"CYC_INT4"	OB 34	OB 34	// Cyclic Interrupt 4
"CYC_INT5"	OB 35	OB 35	// Cyclic Interrupt 5
"HW_INT0"	OB 40	OB 40	// Hardware Interrupt 0
"CYCL_FLT"	OB 80	OB 80	// Cycle Time Fault
"PS_FLT"	OB 81	OB 81	// Power Supply Fault
"I/O_FLT1"	OB 82	OB 82	// I/O Point Fault 1
"CPU_FLT"	OB 84	OB 84	// CPU Fault
"OBNL_FLT"	OB 85	OB 85	// OB Not Loaded Fault
"RACK_FLT"	OB 86	OB 86	// Loss of Rack Fault
"COMM_FLT"	OB 87	OB 87	// Communication Fault
"COMPLETE RESTART"	OB 100	OB 100	// Complete Restart
"PROG_ERR"	OB 121	OB 121	// Programming Error
"MOD_ERR"	OB 122	OB 122	// Module Access Error
"Q0.0"	Q 0.0	BOOL	// Safety Relay Reset
"Q0.1"	Q 0.1	BOOL	// Prestart Sound Alarm
"Q0.2"	Q 0.2	BOOL	// 143BF120C31 - Cmd ON/OFF
"Q0.3"	Q 0.3	BOOL
"Q0.4"	Q 0.4	BOOL
"Q0.5"	Q 0.5	BOOL	// 411SD311C31 - Cmd Open
"Q0.6"	Q 0.6	BOOL	// 411SD321C31 - Cmd Open
"Q0.7"	Q 0.7	BOOL	// 411SD331C31 - Cmd Open
"Q1.0"	Q 1.0	BOOL	// 411SD332C31 - Cmd Open
"Q1.1"	Q 1.1	BOOL	// 411SD333C31 - Cmd Open
"Q1.2"	Q 1.2	BOOL	// 351BV031C31 - Cmd Open
"Q1.3"	Q 1.3	BOOL	// 351BV032C31 - Cmd Open
"Q1.4"	Q 1.4	BOOL	// 351BV033C31 - Cmd Open
"Q1.5"	Q 1.5	BOOL
"Q1.6"	Q 1.6	BOOL	// 351SD141C31 - Cmd Open
"Q1.7"	Q 1.7	BOOL	// 352SD120C31 - Cmd Open
"Q2.0"	Q 2.0	BOOL	// 352SD121C31 - Cmd Open
"Q2.1"	Q 2.1	BOOL
"Q2.2"	Q 2.2	BOOL	// 351SD241C31 - Cmd Open
"Q2.3"	Q 2.3	BOOL	// 352SD220C31 - Cmd Open
"Q2.4"	Q 2.4	BOOL	// 352SD221C31 - Cmd Open
"Q2.5"	Q 2.5	BOOL
"Q2.6"	Q 2.6	BOOL	// 351SD341C31 - Cmd Open
"Q2.7"	Q 2.7	BOOL	// 352SD320C31 - Cmd Open
"Q3.0"	Q 3.0	BOOL	// 352SD321C31 - Cmd Open
"Q3.1"	Q 3.1	BOOL	// 361SD170C31 - Cmd Open
"Q3.2"	Q 3.2	BOOL	// 361SD171C31 - Cmd Open
"Q3.3"	Q 3.3	BOOL	// 361SD172C31 - Cmd Open
"Q3.4"	Q 3.4	BOOL	// 361SD173C31 - Cmd Open
"Q3.5"	Q 3.5	BOOL	// 361SD174C31 - Cmd Open
"Q3.6"	Q 3.6	BOOL	// 361SD175C31 - Cmd Open
"Q3.7"	Q 3.7	BOOL	// 361SD176C31 - Cmd Open
"Q4.0"	Q 4.0	BOOL	// 361SD177C31 - Cmd Open
"Q4.1"	Q 4.1	BOOL	// 411BV151 - Cmd Open
"Q4.2"	Q 4.2	BOOL	// 351SD105C31 - Cmd Open
"Q4.3"	Q 4.3	BOOL	// 351SD106C31 - Cmd Open
"Q4.4"	Q 4.4	BOOL	// 351SD107C31 - Cmd Open
"Q4.5"	Q 4.5	BOOL	// 351SD108C31 - Cmd Open
"Q4.6"	Q 4.6	BOOL	// 351SD109C31 - Cmd Open
"Q4.7"	Q 4.7	BOOL	// 351SD135C31 - Cmd Open
"Q5.0"	Q 5.0	BOOL	// 351SD235C31 - Cmd Open
"Q5.1"	Q 5.1	BOOL	// 351SD335C31 - Cmd Open
"Q5.2"	Q 5.2	BOOL	// SPARE
"Q5.3"	Q 5.3	BOOL	// SPARE
"Q5.4"	Q 5.4	BOOL	// SPARE
"Q5.5"	Q 5.5	BOOL	// SPARE
"Q5.6"	Q 5.6	BOOL	// SPARE
"Q5.7"	Q 5.7	BOOL	// SPARE
"Q6.0"	Q 6.0	BOOL	// SPARE
"Q6.1"	Q 6.1	BOOL	// SPARE
"Q6.2"	Q 6.2	BOOL	// SPARE
"Q6.3"	Q 6.3	BOOL	// SPARE
"Q6.4"	Q 6.4	BOOL	// SPARE
"Q6.5"	Q 6.5	BOOL	// SPARE
"Q6.6"	Q 6.6	BOOL	// SPARE
"Q6.7"	Q 6.7	BOOL	// SPARE
"Q7.0"	Q 7.0	BOOL	// SPARE
"Q7.1"	Q 7.1	BOOL	// SPARE
"Q7.2"	Q 7.2	BOOL	// SPARE
"Q7.3"	Q 7.3	BOOL	// SPARE
"Q7.4"	Q 7.4	BOOL	// SPARE
"Q7.5"	Q 7.5	BOOL	// SPARE
"Q7.6"	Q 7.6	BOOL	// SPARE
"Q7.7"	Q 7.7	BOOL	// SPARE
"Q8.0"	Q 8.0	BOOL	// 351VI110KA1 - Cmd ON/OFF
"Q8.1"	Q 8.1	BOOL	// 351VI210KA1 - Cmd ON/OFF
"Q8.2"	Q 8.2	BOOL	// 351VI310KA1 - Cmd ON/OFF
"Q8.3"	Q 8.3	BOOL	// 352VI110KA1 - Cmd ON/OFF
"Q8.4"	Q 8.4	BOOL	// 352VI111KA1 - Cmd ON/OFF
"Q8.5"	Q 8.5	BOOL	// 352VI210KA1 - Cmd ON/OFF
"Q8.6"	Q 8.6	BOOL	// 352VI211KA1 - Cmd ON/OFF
"Q8.7"	Q 8.7	BOOL	// 352VI310KA1 - Cmd ON/OFF
"Q9.0"	Q 9.0	BOOL	// 352VI311KA1 - Cmd ON/OFF
"Q9.1"	Q 9.1	BOOL	// 341VI201KA1 - Cmd ON/OFF
"Q9.2"	Q 9.2	BOOL	// SPARE
"Q9.3"	Q 9.3	BOOL	// SPARE
"Q9.4"	Q 9.4	BOOL	// SPARE
"Q9.5"	Q 9.5	BOOL	// SPARE
"Q9.6"	Q 9.6	BOOL	// SPARE
"Q9.7"	Q 9.7	BOOL	// SPARE
"Q257.0"	Q 257.0	BOOL	// VAP Pole 1 ON/OFF
"Q261.0"	Q 261.0	BOOL	// VAP Pole 2 ON/OFF
"GET"	SFB 14	SFB 14	// Read Data From a Remote CPU
"PUT"	SFB 15	SFB 15	// Write Data to a Remote CPU
"BLKMOV"	SFC 20	SFC 20	// Copy Variables
"T5"	T 5	TIMER	// BV151 Puls Timer
"GROUP_UDT"	UDT 1	UDT 1
"ROUTE_UDT"	UDT 2	UDT 2
"VAT_SIM"	VAT 1	
"VAT_ANALOG"	VAT 2	
"Filtr"	VAT 3	
"VAT_SIMOCODE"	VAT 4	
"VAT_INPUT"	VAT 5	
"VAT_Weight"	VAT 6	
"VAT_GROUPSIM"	VAT 8	
END_SYMBOL_TABLE
